      "Q776.6" { ExternalVisible := 'False'} : Bool := FALSE;   // Q776.6
      "Q776.7" { ExternalVisible := 'False'} : Bool := FALSE;   // Q776.7
      "Q777.0" { ExternalVisible := 'False'} : Bool := FALSE;   // Q777.0
      "Q777.1" { ExternalVisible := 'False'} : Bool := FALSE;   // Q777.1
      "Q777.2" { ExternalVisible := 'False'} : Bool := FALSE;   // Q777.2
      "Q777.3" { ExternalVisible := 'False'} : Bool := FALSE;   // Q777.3
      "Q777.4" { ExternalVisible := 'False'} : Bool := FALSE;   // Q777.4
      "Q777.5" { ExternalVisible := 'False'} : Bool := FALSE;   // Q777.5
      "Q777.6" { ExternalVisible := 'False'} : Bool := FALSE;   // Q777.6
      "Q777.7" { ExternalVisible := 'False'} : Bool := FALSE;   // Q777.7
      "Q778.0" { ExternalVisible := 'False'} : Bool := FALSE;   // Q778.0
      "Q778.1" { ExternalVisible := 'False'} : Bool := FALSE;   // Q778.1
      "Q778.2" { ExternalVisible := 'False'} : Bool := FALSE;   // Q778.2
      "Q778.3" { ExternalVisible := 'False'} : Bool := FALSE;   // Q778.3
      "Q778.4" { ExternalVisible := 'False'} : Bool := FALSE;   // Q778.4
      "Q778.5" { ExternalVisible := 'False'} : Bool := FALSE;   // Q778.5
      "Q778.6" { ExternalVisible := 'False'} : Bool := FALSE;   // Q778.6
      "Q778.7" { ExternalVisible := 'False'} : Bool := FALSE;   // Q778.7
      "Q779.0" { ExternalVisible := 'False'} : Bool := FALSE;   // Q779.0
      "Q779.1" { ExternalVisible := 'False'} : Bool := FALSE;   // Q779.1
      "Q779.2" { ExternalVisible := 'False'} : Bool := FALSE;   // Q779.2
      "Q779.3" { ExternalVisible := 'False'} : Bool := FALSE;   // Q779.3
      "Q779.4" { ExternalVisible := 'False'} : Bool := FALSE;   // Q779.4
      "Q779.5" { ExternalVisible := 'False'} : Bool := FALSE;   // Q779.5
      "Q779.6" { ExternalVisible := 'False'} : Bool := FALSE;   // Q779.6
      "Q779.7" { ExternalVisible := 'False'} : Bool := FALSE;   // Q779.7
      "Q780.0" { ExternalVisible := 'False'} : Bool := FALSE;   // Q780.0
      "Q780.1" { ExternalVisible := 'False'} : Bool := FALSE;   // Q780.1
      "Q780.2" { ExternalVisible := 'False'} : Bool := FALSE;   // Q780.2
      "Q780.3" { ExternalVisible := 'False'} : Bool := FALSE;   // Q780.3
      "Q780.4" { ExternalVisible := 'False'} : Bool := FALSE;   // Q780.4
      "Q780.5" { ExternalVisible := 'False'} : Bool := FALSE;   // Q780.5
      "Q780.6" { ExternalVisible := 'False'} : Bool := FALSE;   // Q780.6
      "Q780.7" { ExternalVisible := 'False'} : Bool := FALSE;   // Q780.7
      "Q781.0" { ExternalVisible := 'False'} : Bool := FALSE;   // Q781.0
      "Q781.1" { ExternalVisible := 'False'} : Bool := FALSE;   // Q781.1
      "Q781.2" { ExternalVisible := 'False'} : Bool := FALSE;   // Q781.2
      "Q781.3" { ExternalVisible := 'False'} : Bool := FALSE;   // Q781.3
      "Q781.4" { ExternalVisible := 'False'} : Bool := FALSE;   // Q781.4
      "Q781.5" { ExternalVisible := 'False'} : Bool := FALSE;   // Q781.5
      "Q781.6" { ExternalVisible := 'False'} : Bool := FALSE;   // Q781.6
      "Q781.7" { ExternalVisible := 'False'} : Bool := FALSE;   // Q781.7
      "Q782.0" { ExternalVisible := 'False'} : Bool := FALSE;   // Q782.0
      "Q782.1" { ExternalVisible := 'False'} : Bool := FALSE;   // Q782.1
      "Q782.2" { ExternalVisible := 'False'} : Bool := FALSE;   // Q782.2
      "Q782.3" { ExternalVisible := 'False'} : Bool := FALSE;   // Q782.3
      "Q782.4" { ExternalVisible := 'False'} : Bool := FALSE;   // Q782.4
      "Q782.5" { ExternalVisible := 'False'} : Bool := FALSE;   // Q782.5
      "Q782.6" { ExternalVisible := 'False'} : Bool := FALSE;   // Q782.6
      "Q782.7" { ExternalVisible := 'False'} : Bool := FALSE;   // Q782.7
      "Q783.0" { ExternalVisible := 'False'} : Bool := FALSE;   // Q783.0
      "Q783.1" { ExternalVisible := 'False'} : Bool := FALSE;   // Q783.1
      "Q783.2" { ExternalVisible := 'False'} : Bool := FALSE;   // Q783.2
      "Q783.3" { ExternalVisible := 'False'} : Bool := FALSE;   // Q783.3
      "Q783.4" { ExternalVisible := 'False'} : Bool := FALSE;   // Q783.4
      "Q783.5" { ExternalVisible := 'False'} : Bool := FALSE;   // Q783.5
      "Q783.6" { ExternalVisible := 'False'} : Bool := FALSE;   // Q783.6
      "Q783.7" { ExternalVisible := 'False'} : Bool := FALSE;   // Q783.7
      "Q784.0" { ExternalVisible := 'False'} : Bool := FALSE;   // Q784.0
      "Q784.1" { ExternalVisible := 'False'} : Bool := FALSE;   // Q784.1
      "Q784.2" { ExternalVisible := 'False'} : Bool := FALSE;   // Q784.2
      "Q784.3" { ExternalVisible := 'False'} : Bool := FALSE;   // Q784.3
      "Q784.4" { ExternalVisible := 'False'} : Bool := FALSE;   // Q784.4
      "Q784.5" { ExternalVisible := 'False'} : Bool := FALSE;   // Q784.5
      "Q784.6" { ExternalVisible := 'False'} : Bool := FALSE;   // Q784.6
      "Q784.7" { ExternalVisible := 'False'} : Bool := FALSE;   // Q784.7
      "Q785.0" { ExternalVisible := 'False'} : Bool := FALSE;   // Q785.0
      "Q785.1" { ExternalVisible := 'False'} : Bool := FALSE;   // Q785.1
      "Q785.2" { ExternalVisible := 'False'} : Bool := FALSE;   // Q785.2
      "Q785.3" { ExternalVisible := 'False'} : Bool := FALSE;   // Q785.3
      "Q785.4" { ExternalVisible := 'False'} : Bool := FALSE;   // Q785.4
      "Q785.5" { ExternalVisible := 'False'} : Bool := FALSE;   // Q785.5
      "Q785.6" { ExternalVisible := 'False'} : Bool := FALSE;   // Q785.6
      "Q785.7" { ExternalVisible := 'False'} : Bool := FALSE;   // Q785.7
      "Q786.0" { ExternalVisible := 'False'} : Bool := FALSE;   // Q786.0
      "Q786.1" { ExternalVisible := 'False'} : Bool := FALSE;   // Q786.1
      "Q786.2" { ExternalVisible := 'False'} : Bool := FALSE;   // Q786.2
      "Q786.3" { ExternalVisible := 'False'} : Bool := FALSE;   // Q786.3
      "Q786.4" { ExternalVisible := 'False'} : Bool := FALSE;   // Q786.4
      "Q786.5" { ExternalVisible := 'False'} : Bool := FALSE;   // Q786.5
      "Q786.6" { ExternalVisible := 'False'} : Bool := FALSE;   // Q786.6
      "Q786.7" { ExternalVisible := 'False'} : Bool := FALSE;   // Q786.7
      "Q787.0" { ExternalVisible := 'False'} : Bool := FALSE;   // Q787.0
      "Q787.1" { ExternalVisible := 'False'} : Bool := FALSE;   // Q787.1
      "Q787.2" { ExternalVisible := 'False'} : Bool := FALSE;   // Q787.2
      "Q787.3" { ExternalVisible := 'False'} : Bool := FALSE;   // Q787.3
      "Q787.4" { ExternalVisible := 'False'} : Bool := FALSE;   // Q787.4
      "Q787.5" { ExternalVisible := 'False'} : Bool := FALSE;   // Q787.5
      "Q787.6" { ExternalVisible := 'False'} : Bool := FALSE;   // Q787.6
      "Q787.7" { ExternalVisible := 'False'} : Bool := FALSE;   // Q787.7
      "Q788.0" { ExternalVisible := 'False'} : Bool := FALSE;   // Q788.0
      "Q788.1" { ExternalVisible := 'False'} : Bool := FALSE;   // Q788.1
      "Q788.2" { ExternalVisible := 'False'} : Bool := FALSE;   // Q788.2
      "Q788.3" { ExternalVisible := 'False'} : Bool := FALSE;   // Q788.3
      "Q788.4" { ExternalVisible := 'False'} : Bool := FALSE;   // Q788.4
      "Q788.5" { ExternalVisible := 'False'} : Bool := FALSE;   // Q788.5
      "Q788.6" { ExternalVisible := 'False'} : Bool := FALSE;   // Q788.6
      "Q788.7" { ExternalVisible := 'False'} : Bool := FALSE;   // Q788.7
      "Q789.0" { ExternalVisible := 'False'} : Bool := FALSE;   // Q789.0
      "Q789.1" { ExternalVisible := 'False'} : Bool := FALSE;   // Q789.1
      "Q789.2" { ExternalVisible := 'False'} : Bool := FALSE;   // Q789.2
      "Q789.3" { ExternalVisible := 'False'} : Bool := FALSE;   // Q789.3
      "Q789.4" { ExternalVisible := 'False'} : Bool := FALSE;   // Q789.4
      "Q789.5" { ExternalVisible := 'False'} : Bool := FALSE;   // Q789.5
      "Q789.6" { ExternalVisible := 'False'} : Bool := FALSE;   // Q789.6
      "Q789.7" { ExternalVisible := 'False'} : Bool := FALSE;   // Q789.7
      "Q790.0" { ExternalVisible := 'False'} : Bool := FALSE;   // Q790.0
      "Q790.1" { ExternalVisible := 'False'} : Bool := FALSE;   // Q790.1
      "Q790.2" { ExternalVisible := 'False'} : Bool := FALSE;   // Q790.2
      "Q790.3" { ExternalVisible := 'False'} : Bool := FALSE;   // Q790.3
      "Q790.4" { ExternalVisible := 'False'} : Bool := FALSE;   // Q790.4
      "Q790.5" { ExternalVisible := 'False'} : Bool := FALSE;   // Q790.5
      "Q790.6" { ExternalVisible := 'False'} : Bool := FALSE;   // Q790.6
      "Q790.7" { ExternalVisible := 'False'} : Bool := FALSE;   // Q790.7
      "Q791.0" { ExternalVisible := 'False'} : Bool := FALSE;   // Q791.0
      "Q791.1" { ExternalVisible := 'False'} : Bool := FALSE;   // Q791.1
      "Q791.2" { ExternalVisible := 'False'} : Bool := FALSE;   // Q791.2
      "Q791.3" { ExternalVisible := 'False'} : Bool := FALSE;   // Q791.3
      "Q791.4" { ExternalVisible := 'False'} : Bool := FALSE;   // Q791.4
      "Q791.5" { ExternalVisible := 'False'} : Bool := FALSE;   // Q791.5
      "Q791.6" { ExternalVisible := 'False'} : Bool := FALSE;   // Q791.6
      "Q791.7" { ExternalVisible := 'False'} : Bool := FALSE;   // Q791.7
      "Q792.0" { ExternalVisible := 'False'} : Bool := FALSE;   // Q792.0
      "Q792.1" { ExternalVisible := 'False'} : Bool := FALSE;   // Q792.1
      "Q792.2" { ExternalVisible := 'False'} : Bool := FALSE;   // Q792.2
      "Q792.3" { ExternalVisible := 'False'} : Bool := FALSE;   // Q792.3
      "Q792.4" { ExternalVisible := 'False'} : Bool := FALSE;   // Q792.4
      "Q792.5" { ExternalVisible := 'False'} : Bool := FALSE;   // Q792.5
      "Q792.6" { ExternalVisible := 'False'} : Bool := FALSE;   // Q792.6
      "Q792.7" { ExternalVisible := 'False'} : Bool := FALSE;   // Q792.7
      "Q793.0" { ExternalVisible := 'False'} : Bool := FALSE;   // Q793.0
      "Q793.1" { ExternalVisible := 'False'} : Bool := FALSE;   // Q793.1
      "Q793.2" { ExternalVisible := 'False'} : Bool := FALSE;   // Q793.2
      "Q793.3" { ExternalVisible := 'False'} : Bool := FALSE;   // Q793.3
      "Q793.4" { ExternalVisible := 'False'} : Bool := FALSE;   // Q793.4
      "Q793.5" { ExternalVisible := 'False'} : Bool := FALSE;   // Q793.5
      "Q793.6" { ExternalVisible := 'False'} : Bool := FALSE;   // Q793.6
      "Q793.7" { ExternalVisible := 'False'} : Bool := FALSE;   // Q793.7
      "Q794.0" { ExternalVisible := 'False'} : Bool := FALSE;   // Q794.0
      "Q794.1" { ExternalVisible := 'False'} : Bool := FALSE;   // Q794.1
      "Q794.2" { ExternalVisible := 'False'} : Bool := FALSE;   // Q794.2
      "Q794.3" { ExternalVisible := 'False'} : Bool := FALSE;   // Q794.3
      "Q794.4" { ExternalVisible := 'False'} : Bool := FALSE;   // Q794.4
      "Q794.5" { ExternalVisible := 'False'} : Bool := FALSE;   // Q794.5
      "Q794.6" { ExternalVisible := 'False'} : Bool := FALSE;   // Q794.6
      "Q794.7" { ExternalVisible := 'False'} : Bool := FALSE;   // Q794.7
      "Q795.0" { ExternalVisible := 'False'} : Bool := FALSE;   // Q795.0
      "Q795.1" { ExternalVisible := 'False'} : Bool := FALSE;   // Q795.1
      "Q795.2" { ExternalVisible := 'False'} : Bool := FALSE;   // Q795.2
      "Q795.3" { ExternalVisible := 'False'} : Bool := FALSE;   // Q795.3
      "Q795.4" { ExternalVisible := 'False'} : Bool := FALSE;   // Q795.4
      "Q795.5" { ExternalVisible := 'False'} : Bool := FALSE;   // Q795.5
      "Q795.6" { ExternalVisible := 'False'} : Bool := FALSE;   // Q795.6
      "Q795.7" { ExternalVisible := 'False'} : Bool := FALSE;   // Q795.7
      "Q796.0" { ExternalVisible := 'False'} : Bool := FALSE;   // Q796.0
      "Q796.1" { ExternalVisible := 'False'} : Bool := FALSE;   // Q796.1
      "Q796.2" { ExternalVisible := 'False'} : Bool := FALSE;   // Q796.2
      "Q796.3" { ExternalVisible := 'False'} : Bool := FALSE;   // Q796.3
      "Q796.4" { ExternalVisible := 'False'} : Bool := FALSE;   // Q796.4
      "Q796.5" { ExternalVisible := 'False'} : Bool := FALSE;   // Q796.5
      "Q796.6" { ExternalVisible := 'False'} : Bool := FALSE;   // Q796.6
      "Q796.7" { ExternalVisible := 'False'} : Bool := FALSE;   // Q796.7
      "Q797.0" { ExternalVisible := 'False'} : Bool := FALSE;   // Q797.0
      "Q797.1" { ExternalVisible := 'False'} : Bool := FALSE;   // Q797.1
      "Q797.2" { ExternalVisible := 'False'} : Bool := FALSE;   // Q797.2
      "Q797.3" { ExternalVisible := 'False'} : Bool := FALSE;   // Q797.3
      "Q797.4" { ExternalVisible := 'False'} : Bool := FALSE;   // Q797.4
      "Q797.5" { ExternalVisible := 'False'} : Bool := FALSE;   // Q797.5
      "Q797.6" { ExternalVisible := 'False'} : Bool := FALSE;   // Q797.6
      "Q797.7" { ExternalVisible := 'False'} : Bool := FALSE;   // Q797.7
      "Q798.0" { ExternalVisible := 'False'} : Bool := FALSE;   // Q798.0
      "Q798.1" { ExternalVisible := 'False'} : Bool := FALSE;   // Q798.1
      "Q798.2" { ExternalVisible := 'False'} : Bool := FALSE;   // Q798.2
      "Q798.3" { ExternalVisible := 'False'} : Bool := FALSE;   // Q798.3
      "Q798.4" { ExternalVisible := 'False'} : Bool := FALSE;   // Q798.4
      "Q798.5" { ExternalVisible := 'False'} : Bool := FALSE;   // Q798.5
      "Q798.6" { ExternalVisible := 'False'} : Bool := FALSE;   // Q798.6
      "Q798.7" { ExternalVisible := 'False'} : Bool := FALSE;   // Q798.7
      "Q799.0" { ExternalVisible := 'False'} : Bool := FALSE;   // Q799.0
      "Q799.1" { ExternalVisible := 'False'} : Bool := FALSE;   // Q799.1
      "Q799.2" { ExternalVisible := 'False'} : Bool := FALSE;   // Q799.2
      "Q799.3" { ExternalVisible := 'False'} : Bool := FALSE;   // Q799.3
      "Q799.4" { ExternalVisible := 'False'} : Bool := FALSE;   // Q799.4
      "Q799.5" { ExternalVisible := 'False'} : Bool := FALSE;   // Q799.5
      "Q799.6" { ExternalVisible := 'False'} : Bool := FALSE;   // Q799.6
      "Q799.7" { ExternalVisible := 'False'} : Bool := FALSE;   // Q799.7
      "Q800.0" { ExternalVisible := 'False'} : Bool := FALSE;   // Q800.0
      "Q800.1" { ExternalVisible := 'False'} : Bool := FALSE;   // Q800.1
      "Q800.2" { ExternalVisible := 'False'} : Bool := FALSE;   // Q800.2
      "Q800.3" { ExternalVisible := 'False'} : Bool := FALSE;   // Q800.3
      "Q800.4" { ExternalVisible := 'False'} : Bool := FALSE;   // Q800.4
      "Q800.5" { ExternalVisible := 'False'} : Bool := FALSE;   // Q800.5
      "Q800.6" { ExternalVisible := 'False'} : Bool := FALSE;   // Q800.6
      "Q800.7" { ExternalVisible := 'False'} : Bool := FALSE;   // Q800.7
      "Q801.0" { ExternalVisible := 'False'} : Bool := FALSE;   // Q801.0
      "Q801.1" { ExternalVisible := 'False'} : Bool := FALSE;   // Q801.1
      "Q801.2" { ExternalVisible := 'False'} : Bool := FALSE;   // Q801.2
      "Q801.3" { ExternalVisible := 'False'} : Bool := FALSE;   // Q801.3
      "Q801.4" { ExternalVisible := 'False'} : Bool := FALSE;   // Q801.4
      "Q801.5" { ExternalVisible := 'False'} : Bool := FALSE;   // Q801.5
      "Q801.6" { ExternalVisible := 'False'} : Bool := FALSE;   // Q801.6
      "Q801.7" { ExternalVisible := 'False'} : Bool := FALSE;   // Q801.7
      "Q802.0" { ExternalVisible := 'False'} : Bool := FALSE;   // Q802.0
      "Q802.1" { ExternalVisible := 'False'} : Bool := FALSE;   // Q802.1
      "Q802.2" { ExternalVisible := 'False'} : Bool := FALSE;   // Q802.2
      "Q802.3" { ExternalVisible := 'False'} : Bool := FALSE;   // Q802.3
      "Q802.4" { ExternalVisible := 'False'} : Bool := FALSE;   // Q802.4
      "Q802.5" { ExternalVisible := 'False'} : Bool := FALSE;   // Q802.5
      "Q802.6" { ExternalVisible := 'False'} : Bool := FALSE;   // Q802.6
      "Q802.7" { ExternalVisible := 'False'} : Bool := FALSE;   // Q802.7
      "Q803.0" { ExternalVisible := 'False'} : Bool := FALSE;   // Q803.0
      "Q803.1" { ExternalVisible := 'False'} : Bool := FALSE;   // Q803.1
      "Q803.2" { ExternalVisible := 'False'} : Bool := FALSE;   // Q803.2
      "Q803.3" { ExternalVisible := 'False'} : Bool := FALSE;   // Q803.3
      "Q803.4" { ExternalVisible := 'False'} : Bool := FALSE;   // Q803.4
      "Q803.5" { ExternalVisible := 'False'} : Bool := FALSE;   // Q803.5
      "Q803.6" { ExternalVisible := 'False'} : Bool := FALSE;   // Q803.6
      "Q803.7" { ExternalVisible := 'False'} : Bool := FALSE;   // Q803.7
      "Q804.0" { ExternalVisible := 'False'} : Bool := FALSE;   // Q804.0
      "Q804.1" { ExternalVisible := 'False'} : Bool := FALSE;   // Q804.1
      "Q804.2" { ExternalVisible := 'False'} : Bool := FALSE;   // Q804.2
      "Q804.3" { ExternalVisible := 'False'} : Bool := FALSE;   // Q804.3
      "Q804.4" { ExternalVisible := 'False'} : Bool := FALSE;   // Q804.4
      "Q804.5" { ExternalVisible := 'False'} : Bool := FALSE;   // Q804.5
      "Q804.6" { ExternalVisible := 'False'} : Bool := FALSE;   // Q804.6
      "Q804.7" { ExternalVisible := 'False'} : Bool := FALSE;   // Q804.7
      "Q805.0" { ExternalVisible := 'False'} : Bool := FALSE;   // Q805.0
      "Q805.1" { ExternalVisible := 'False'} : Bool := FALSE;   // Q805.1
      "Q805.2" { ExternalVisible := 'False'} : Bool := FALSE;   // Q805.2
      "Q805.3" { ExternalVisible := 'False'} : Bool := FALSE;   // Q805.3
      "Q805.4" { ExternalVisible := 'False'} : Bool := FALSE;   // Q805.4
      "Q805.5" { ExternalVisible := 'False'} : Bool := FALSE;   // Q805.5
      "Q805.6" { ExternalVisible := 'False'} : Bool := FALSE;   // Q805.6
      "Q805.7" { ExternalVisible := 'False'} : Bool := FALSE;   // Q805.7
      "Q806.0" { ExternalVisible := 'False'} : Bool := FALSE;   // Q806.0
      "Q806.1" { ExternalVisible := 'False'} : Bool := FALSE;   // Q806.1
      "Q806.2" { ExternalVisible := 'False'} : Bool := FALSE;   // Q806.2
      "Q806.3" { ExternalVisible := 'False'} : Bool := FALSE;   // Q806.3
      "Q806.4" { ExternalVisible := 'False'} : Bool := FALSE;   // Q806.4
      "Q806.5" { ExternalVisible := 'False'} : Bool := FALSE;   // Q806.5
      "Q806.6" { ExternalVisible := 'False'} : Bool := FALSE;   // Q806.6
      "Q806.7" { ExternalVisible := 'False'} : Bool := FALSE;   // Q806.7
      "Q807.0" { ExternalVisible := 'False'} : Bool := FALSE;   // Q807.0
      "Q807.1" { ExternalVisible := 'False'} : Bool := FALSE;   // Q807.1
      "Q807.2" { ExternalVisible := 'False'} : Bool := FALSE;   // Q807.2
      "Q807.3" { ExternalVisible := 'False'} : Bool := FALSE;   // Q807.3
      "Q807.4" { ExternalVisible := 'False'} : Bool := FALSE;   // Q807.4
      "Q807.5" { ExternalVisible := 'False'} : Bool := FALSE;   // Q807.5
      "Q807.6" { ExternalVisible := 'False'} : Bool := FALSE;   // Q807.6
      "Q807.7" { ExternalVisible := 'False'} : Bool := FALSE;   // Q807.7
      "Q808.0" { ExternalVisible := 'False'} : Bool := FALSE;   // Q808.0
      "Q808.1" { ExternalVisible := 'False'} : Bool := FALSE;   // Q808.1
      "Q808.2" { ExternalVisible := 'False'} : Bool := FALSE;   // Q808.2
      "Q808.3" { ExternalVisible := 'False'} : Bool := FALSE;   // Q808.3
      "Q808.4" { ExternalVisible := 'False'} : Bool := FALSE;   // Q808.4
      "Q808.5" { ExternalVisible := 'False'} : Bool := FALSE;   // Q808.5
      "Q808.6" { ExternalVisible := 'False'} : Bool := FALSE;   // Q808.6
      "Q808.7" { ExternalVisible := 'False'} : Bool := FALSE;   // Q808.7
      "Q809.0" { ExternalVisible := 'False'} : Bool := FALSE;   // Q809.0
      "Q809.1" { ExternalVisible := 'False'} : Bool := FALSE;   // Q809.1
      "Q809.2" { ExternalVisible := 'False'} : Bool := FALSE;   // Q809.2
      "Q809.3" { ExternalVisible := 'False'} : Bool := FALSE;   // Q809.3
      "Q809.4" { ExternalVisible := 'False'} : Bool := FALSE;   // Q809.4
      "Q809.5" { ExternalVisible := 'False'} : Bool := FALSE;   // Q809.5
      "Q809.6" { ExternalVisible := 'False'} : Bool := FALSE;   // Q809.6
      "Q809.7" { ExternalVisible := 'False'} : Bool := FALSE;   // Q809.7
      "Q810.0" { ExternalVisible := 'False'} : Bool := FALSE;   // Q810.0
      "Q810.1" { ExternalVisible := 'False'} : Bool := FALSE;   // Q810.1
      "Q810.2" { ExternalVisible := 'False'} : Bool := FALSE;   // Q810.2
      "Q810.3" { ExternalVisible := 'False'} : Bool := FALSE;   // Q810.3
      "Q810.4" { ExternalVisible := 'False'} : Bool := FALSE;   // Q810.4
      "Q810.5" { ExternalVisible := 'False'} : Bool := FALSE;   // Q810.5
      "Q810.6" { ExternalVisible := 'False'} : Bool := FALSE;   // Q810.6
      "Q810.7" { ExternalVisible := 'False'} : Bool := FALSE;   // Q810.7
      "Q811.0" { ExternalVisible := 'False'} : Bool := FALSE;   // Q811.0
      "Q811.1" { ExternalVisible := 'False'} : Bool := FALSE;   // Q811.1
      "Q811.2" { ExternalVisible := 'False'} : Bool := FALSE;   // Q811.2
      "Q811.3" { ExternalVisible := 'False'} : Bool := FALSE;   // Q811.3
      "Q811.4" { ExternalVisible := 'False'} : Bool := FALSE;   // Q811.4
      "Q811.5" { ExternalVisible := 'False'} : Bool := FALSE;   // Q811.5
      "Q811.6" { ExternalVisible := 'False'} : Bool := FALSE;   // Q811.6
      "Q811.7" { ExternalVisible := 'False'} : Bool := FALSE;   // Q811.7
      "Q812.0" { ExternalVisible := 'False'} : Bool := FALSE;   // Q812.0
      "Q812.1" { ExternalVisible := 'False'} : Bool := FALSE;   // Q812.1
      "Q812.2" { ExternalVisible := 'False'} : Bool := FALSE;   // Q812.2
      "Q812.3" { ExternalVisible := 'False'} : Bool := FALSE;   // Q812.3
      "Q812.4" { ExternalVisible := 'False'} : Bool := FALSE;   // Q812.4
      "Q812.5" { ExternalVisible := 'False'} : Bool := FALSE;   // Q812.5
      "Q812.6" { ExternalVisible := 'False'} : Bool := FALSE;   // Q812.6
      "Q812.7" { ExternalVisible := 'False'} : Bool := FALSE;   // Q812.7
      "Q813.0" { ExternalVisible := 'False'} : Bool := FALSE;   // Q813.0
      "Q813.1" { ExternalVisible := 'False'} : Bool := FALSE;   // Q813.1
      "Q813.2" { ExternalVisible := 'False'} : Bool := FALSE;   // Q813.2
      "Q813.3" { ExternalVisible := 'False'} : Bool := FALSE;   // Q813.3
      "Q813.4" { ExternalVisible := 'False'} : Bool := FALSE;   // Q813.4
      "Q813.5" { ExternalVisible := 'False'} : Bool := FALSE;   // Q813.5
      "Q813.6" { ExternalVisible := 'False'} : Bool := FALSE;   // Q813.6
      "Q813.7" { ExternalVisible := 'False'} : Bool := FALSE;   // Q813.7
      "Q814.0" { ExternalVisible := 'False'} : Bool := FALSE;   // Q814.0
      "Q814.1" { ExternalVisible := 'False'} : Bool := FALSE;   // Q814.1
      "Q814.2" { ExternalVisible := 'False'} : Bool := FALSE;   // Q814.2
      "Q814.3" { ExternalVisible := 'False'} : Bool := FALSE;   // Q814.3
      "Q814.4" { ExternalVisible := 'False'} : Bool := FALSE;   // Q814.4
      "Q814.5" { ExternalVisible := 'False'} : Bool := FALSE;   // Q814.5
      "Q814.6" { ExternalVisible := 'False'} : Bool := FALSE;   // Q814.6
      "Q814.7" { ExternalVisible := 'False'} : Bool := FALSE;   // Q814.7
      "Q815.0" { ExternalVisible := 'False'} : Bool := FALSE;   // Q815.0
      "Q815.1" { ExternalVisible := 'False'} : Bool := FALSE;   // Q815.1
      "Q815.2" { ExternalVisible := 'False'} : Bool := FALSE;   // Q815.2
      "Q815.3" { ExternalVisible := 'False'} : Bool := FALSE;   // Q815.3
      "Q815.4" { ExternalVisible := 'False'} : Bool := FALSE;   // Q815.4
      "Q815.5" { ExternalVisible := 'False'} : Bool := FALSE;   // Q815.5
      "Q815.6" { ExternalVisible := 'False'} : Bool := FALSE;   // Q815.6
      "Q815.7" { ExternalVisible := 'False'} : Bool := FALSE;   // Q815.7
      "Q816.0" { ExternalVisible := 'False'} : Bool := FALSE;   // Q816.0
      "Q816.1" { ExternalVisible := 'False'} : Bool := FALSE;   // Q816.1
      "Q816.2" { ExternalVisible := 'False'} : Bool := FALSE;   // Q816.2
      "Q816.3" { ExternalVisible := 'False'} : Bool := FALSE;   // Q816.3
      "Q816.4" { ExternalVisible := 'False'} : Bool := FALSE;   // Q816.4
      "Q816.5" { ExternalVisible := 'False'} : Bool := FALSE;   // Q816.5
      "Q816.6" { ExternalVisible := 'False'} : Bool := FALSE;   // Q816.6
      "Q816.7" { ExternalVisible := 'False'} : Bool := FALSE;   // Q816.7
      "Q817.0" { ExternalVisible := 'False'} : Bool := FALSE;   // Q817.0
      "Q817.1" { ExternalVisible := 'False'} : Bool := FALSE;   // Q817.1
      "Q817.2" { ExternalVisible := 'False'} : Bool := FALSE;   // Q817.2
      "Q817.3" { ExternalVisible := 'False'} : Bool := FALSE;   // Q817.3
      "Q817.4" { ExternalVisible := 'False'} : Bool := FALSE;   // Q817.4
      "Q817.5" { ExternalVisible := 'False'} : Bool := FALSE;   // Q817.5
      "Q817.6" { ExternalVisible := 'False'} : Bool := FALSE;   // Q817.6
      "Q817.7" { ExternalVisible := 'False'} : Bool := FALSE;   // Q817.7
      "Q818.0" { ExternalVisible := 'False'} : Bool := FALSE;   // Q818.0
      "Q818.1" { ExternalVisible := 'False'} : Bool := FALSE;   // Q818.1
      "Q818.2" { ExternalVisible := 'False'} : Bool := FALSE;   // Q818.2
      "Q818.3" { ExternalVisible := 'False'} : Bool := FALSE;   // Q818.3
      "Q818.4" { ExternalVisible := 'False'} : Bool := FALSE;   // Q818.4
      "Q818.5" { ExternalVisible := 'False'} : Bool := FALSE;   // Q818.5
      "Q818.6" { ExternalVisible := 'False'} : Bool := FALSE;   // Q818.6
      "Q818.7" { ExternalVisible := 'False'} : Bool := FALSE;   // Q818.7
      "Q819.0" { ExternalVisible := 'False'} : Bool := FALSE;   // Q819.0
      "Q819.1" { ExternalVisible := 'False'} : Bool := FALSE;   // Q819.1
      "Q819.2" { ExternalVisible := 'False'} : Bool := FALSE;   // Q819.2
      "Q819.3" { ExternalVisible := 'False'} : Bool := FALSE;   // Q819.3
      "Q819.4" { ExternalVisible := 'False'} : Bool := FALSE;   // Q819.4
      "Q819.5" { ExternalVisible := 'False'} : Bool := FALSE;   // Q819.5
      "Q819.6" { ExternalVisible := 'False'} : Bool := FALSE;   // Q819.6
      "Q819.7" { ExternalVisible := 'False'} : Bool := FALSE;   // Q819.7
      "Q820.0" { ExternalVisible := 'False'} : Bool := FALSE;   // Q820.0
      "Q820.1" { ExternalVisible := 'False'} : Bool := FALSE;   // Q820.1
      "Q820.2" { ExternalVisible := 'False'} : Bool := FALSE;   // Q820.2
      "Q820.3" { ExternalVisible := 'False'} : Bool := FALSE;   // Q820.3
      "Q820.4" { ExternalVisible := 'False'} : Bool := FALSE;   // Q820.4
      "Q820.5" { ExternalVisible := 'False'} : Bool := FALSE;   // Q820.5
      "Q820.6" { ExternalVisible := 'False'} : Bool := FALSE;   // Q820.6
      "Q820.7" { ExternalVisible := 'False'} : Bool := FALSE;   // Q820.7
      "Q821.0" { ExternalVisible := 'False'} : Bool := FALSE;   // Q821.0
      "Q821.1" { ExternalVisible := 'False'} : Bool := FALSE;   // Q821.1
      "Q821.2" { ExternalVisible := 'False'} : Bool := FALSE;   // Q821.2
      "Q821.3" { ExternalVisible := 'False'} : Bool := FALSE;   // Q821.3
      "Q821.4" { ExternalVisible := 'False'} : Bool := FALSE;   // Q821.4
      "Q821.5" { ExternalVisible := 'False'} : Bool := FALSE;   // Q821.5
      "Q821.6" { ExternalVisible := 'False'} : Bool := FALSE;   // Q821.6
      "Q821.7" { ExternalVisible := 'False'} : Bool := FALSE;   // Q821.7
      "Q822.0" { ExternalVisible := 'False'} : Bool := FALSE;   // Q822.0
      "Q822.1" { ExternalVisible := 'False'} : Bool := FALSE;   // Q822.1
      "Q822.2" { ExternalVisible := 'False'} : Bool := FALSE;   // Q822.2
      "Q822.3" { ExternalVisible := 'False'} : Bool := FALSE;   // Q822.3
      "Q822.4" { ExternalVisible := 'False'} : Bool := FALSE;   // Q822.4
      "Q822.5" { ExternalVisible := 'False'} : Bool := FALSE;   // Q822.5
      "Q822.6" { ExternalVisible := 'False'} : Bool := FALSE;   // Q822.6
      "Q822.7" { ExternalVisible := 'False'} : Bool := FALSE;   // Q822.7
      "Q823.0" { ExternalVisible := 'False'} : Bool := FALSE;   // Q823.0
      "Q823.1" { ExternalVisible := 'False'} : Bool := FALSE;   // Q823.1
      "Q823.2" { ExternalVisible := 'False'} : Bool := FALSE;   // Q823.2
      "Q823.3" { ExternalVisible := 'False'} : Bool := FALSE;   // Q823.3
      "Q823.4" { ExternalVisible := 'False'} : Bool := FALSE;   // Q823.4
      "Q823.5" { ExternalVisible := 'False'} : Bool := FALSE;   // Q823.5
      "Q823.6" { ExternalVisible := 'False'} : Bool := FALSE;   // Q823.6
      "Q823.7" { ExternalVisible := 'False'} : Bool := FALSE;   // Q823.7
      "Q824.0" { ExternalVisible := 'False'} : Bool := FALSE;   // Q824.0
      "Q824.1" { ExternalVisible := 'False'} : Bool := FALSE;   // Q824.1
      "Q824.2" { ExternalVisible := 'False'} : Bool := FALSE;   // Q824.2
      "Q824.3" { ExternalVisible := 'False'} : Bool := FALSE;   // Q824.3
      "Q824.4" { ExternalVisible := 'False'} : Bool := FALSE;   // Q824.4
      "Q824.5" { ExternalVisible := 'False'} : Bool := FALSE;   // Q824.5
      "Q824.6" { ExternalVisible := 'False'} : Bool := FALSE;   // Q824.6
      "Q824.7" { ExternalVisible := 'False'} : Bool := FALSE;   // Q824.7
      "Q825.0" { ExternalVisible := 'False'} : Bool := FALSE;   // Q825.0
      "Q825.1" { ExternalVisible := 'False'} : Bool := FALSE;   // Q825.1
      "Q825.2" { ExternalVisible := 'False'} : Bool := FALSE;   // Q825.2
      "Q825.3" { ExternalVisible := 'False'} : Bool := FALSE;   // Q825.3
      "Q825.4" { ExternalVisible := 'False'} : Bool := FALSE;   // Q825.4
      "Q825.5" { ExternalVisible := 'False'} : Bool := FALSE;   // Q825.5
      "Q825.6" { ExternalVisible := 'False'} : Bool := FALSE;   // Q825.6
      "Q825.7" { ExternalVisible := 'False'} : Bool := FALSE;   // Q825.7
      "Q826.0" { ExternalVisible := 'False'} : Bool := FALSE;   // Q826.0
      "Q826.1" { ExternalVisible := 'False'} : Bool := FALSE;   // Q826.1
      "Q826.2" { ExternalVisible := 'False'} : Bool := FALSE;   // Q826.2
      "Q826.3" { ExternalVisible := 'False'} : Bool := FALSE;   // Q826.3
      "Q826.4" { ExternalVisible := 'False'} : Bool := FALSE;   // Q826.4
      "Q826.5" { ExternalVisible := 'False'} : Bool := FALSE;   // Q826.5
      "Q826.6" { ExternalVisible := 'False'} : Bool := FALSE;   // Q826.6
      "Q826.7" { ExternalVisible := 'False'} : Bool := FALSE;   // Q826.7
      "Q827.0" { ExternalVisible := 'False'} : Bool := FALSE;   // Q827.0
      "Q827.1" { ExternalVisible := 'False'} : Bool := FALSE;   // Q827.1
      "Q827.2" { ExternalVisible := 'False'} : Bool := FALSE;   // Q827.2
      "Q827.3" { ExternalVisible := 'False'} : Bool := FALSE;   // Q827.3
      "Q827.4" { ExternalVisible := 'False'} : Bool := FALSE;   // Q827.4
      "Q827.5" { ExternalVisible := 'False'} : Bool := FALSE;   // Q827.5
      "Q827.6" { ExternalVisible := 'False'} : Bool := FALSE;   // Q827.6
      "Q827.7" { ExternalVisible := 'False'} : Bool := FALSE;   // Q827.7
      "Q828.0" { ExternalVisible := 'False'} : Bool := FALSE;   // Q828.0
      "Q828.1" { ExternalVisible := 'False'} : Bool := FALSE;   // Q828.1
      "Q828.2" { ExternalVisible := 'False'} : Bool := FALSE;   // Q828.2
      "Q828.3" { ExternalVisible := 'False'} : Bool := FALSE;   // Q828.3
      "Q828.4" { ExternalVisible := 'False'} : Bool := FALSE;   // Q828.4
      "Q828.5" { ExternalVisible := 'False'} : Bool := FALSE;   // Q828.5
      "Q828.6" { ExternalVisible := 'False'} : Bool := FALSE;   // Q828.6
      "Q828.7" { ExternalVisible := 'False'} : Bool := FALSE;   // Q828.7
      "Q829.0" { ExternalVisible := 'False'} : Bool := FALSE;   // Q829.0
      "Q829.1" { ExternalVisible := 'False'} : Bool := FALSE;   // Q829.1
      "Q829.2" { ExternalVisible := 'False'} : Bool := FALSE;   // Q829.2
      "Q829.3" { ExternalVisible := 'False'} : Bool := FALSE;   // Q829.3
      "Q829.4" { ExternalVisible := 'False'} : Bool := FALSE;   // Q829.4
      "Q829.5" { ExternalVisible := 'False'} : Bool := FALSE;   // Q829.5
      "Q829.6" { ExternalVisible := 'False'} : Bool := FALSE;   // Q829.6
      "Q829.7" { ExternalVisible := 'False'} : Bool := FALSE;   // Q829.7
      "Q830.0" { ExternalVisible := 'False'} : Bool := FALSE;   // Q830.0
      "Q830.1" { ExternalVisible := 'False'} : Bool := FALSE;   // Q830.1
      "Q830.2" { ExternalVisible := 'False'} : Bool := FALSE;   // Q830.2
      "Q830.3" { ExternalVisible := 'False'} : Bool := FALSE;   // Q830.3
      "Q830.4" { ExternalVisible := 'False'} : Bool := FALSE;   // Q830.4
      "Q830.5" { ExternalVisible := 'False'} : Bool := FALSE;   // Q830.5
      "Q830.6" { ExternalVisible := 'False'} : Bool := FALSE;   // Q830.6
      "Q830.7" { ExternalVisible := 'False'} : Bool := FALSE;   // Q830.7
      "Q831.0" { ExternalVisible := 'False'} : Bool := FALSE;   // Q831.0
      "Q831.1" { ExternalVisible := 'False'} : Bool := FALSE;   // Q831.1
      "Q831.2" { ExternalVisible := 'False'} : Bool := FALSE;   // Q831.2
      "Q831.3" { ExternalVisible := 'False'} : Bool := FALSE;   // Q831.3
      "Q831.4" { ExternalVisible := 'False'} : Bool := FALSE;   // Q831.4
      "Q831.5" { ExternalVisible := 'False'} : Bool := FALSE;   // Q831.5
      "Q831.6" { ExternalVisible := 'False'} : Bool := FALSE;   // Q831.6
      "Q831.7" { ExternalVisible := 'False'} : Bool := FALSE;   // Q831.7
      "Q832.0" { ExternalVisible := 'False'} : Bool := FALSE;   // Q832.0
      "Q832.1" { ExternalVisible := 'False'} : Bool := FALSE;   // Q832.1
      "Q832.2" { ExternalVisible := 'False'} : Bool := FALSE;   // Q832.2
      "Q832.3" { ExternalVisible := 'False'} : Bool := FALSE;   // Q832.3
      "Q832.4" { ExternalVisible := 'False'} : Bool := FALSE;   // Q832.4
      "Q832.5" { ExternalVisible := 'False'} : Bool := FALSE;   // Q832.5
      "Q832.6" { ExternalVisible := 'False'} : Bool := FALSE;   // Q832.6
      "Q832.7" { ExternalVisible := 'False'} : Bool := FALSE;   // Q832.7
      "Q833.0" { ExternalVisible := 'False'} : Bool := FALSE;   // Q833.0
      "Q833.1" { ExternalVisible := 'False'} : Bool := FALSE;   // Q833.1
      "Q833.2" { ExternalVisible := 'False'} : Bool := FALSE;   // Q833.2
      "Q833.3" { ExternalVisible := 'False'} : Bool := FALSE;   // Q833.3
      "Q833.4" { ExternalVisible := 'False'} : Bool := FALSE;   // Q833.4
      "Q833.5" { ExternalVisible := 'False'} : Bool := FALSE;   // Q833.5
      "Q833.6" { ExternalVisible := 'False'} : Bool := FALSE;   // Q833.6
      "Q833.7" { ExternalVisible := 'False'} : Bool := FALSE;   // Q833.7
      "Q834.0" { ExternalVisible := 'False'} : Bool := FALSE;   // Q834.0
      "Q834.1" { ExternalVisible := 'False'} : Bool := FALSE;   // Q834.1
      "Q834.2" { ExternalVisible := 'False'} : Bool := FALSE;   // Q834.2
      "Q834.3" { ExternalVisible := 'False'} : Bool := FALSE;   // Q834.3
      "Q834.4" { ExternalVisible := 'False'} : Bool := FALSE;   // Q834.4
      "Q834.5" { ExternalVisible := 'False'} : Bool := FALSE;   // Q834.5
      "Q834.6" { ExternalVisible := 'False'} : Bool := FALSE;   // Q834.6
      "Q834.7" { ExternalVisible := 'False'} : Bool := FALSE;   // Q834.7
      "Q835.0" { ExternalVisible := 'False'} : Bool := FALSE;   // Q835.0
      "Q835.1" { ExternalVisible := 'False'} : Bool := FALSE;   // Q835.1
      "Q835.2" { ExternalVisible := 'False'} : Bool := FALSE;   // Q835.2
      "Q835.3" { ExternalVisible := 'False'} : Bool := FALSE;   // Q835.3
      "Q835.4" { ExternalVisible := 'False'} : Bool := FALSE;   // Q835.4
      "Q835.5" { ExternalVisible := 'False'} : Bool := FALSE;   // Q835.5
      "Q835.6" { ExternalVisible := 'False'} : Bool := FALSE;   // Q835.6
      "Q835.7" { ExternalVisible := 'False'} : Bool := FALSE;   // Q835.7
      "Q836.0" { ExternalVisible := 'False'} : Bool := FALSE;   // Q836.0
      "Q836.1" { ExternalVisible := 'False'} : Bool := FALSE;   // Q836.1
      "Q836.2" { ExternalVisible := 'False'} : Bool := FALSE;   // Q836.2
      "Q836.3" { ExternalVisible := 'False'} : Bool := FALSE;   // Q836.3
      "Q836.4" { ExternalVisible := 'False'} : Bool := FALSE;   // Q836.4
      "Q836.5" { ExternalVisible := 'False'} : Bool := FALSE;   // Q836.5
      "Q836.6" { ExternalVisible := 'False'} : Bool := FALSE;   // Q836.6
      "Q836.7" { ExternalVisible := 'False'} : Bool := FALSE;   // Q836.7
      "Q837.0" { ExternalVisible := 'False'} : Bool := FALSE;   // Q837.0
      "Q837.1" { ExternalVisible := 'False'} : Bool := FALSE;   // Q837.1
      "Q837.2" { ExternalVisible := 'False'} : Bool := FALSE;   // Q837.2
      "Q837.3" { ExternalVisible := 'False'} : Bool := FALSE;   // Q837.3
      "Q837.4" { ExternalVisible := 'False'} : Bool := FALSE;   // Q837.4
      "Q837.5" { ExternalVisible := 'False'} : Bool := FALSE;   // Q837.5
      "Q837.6" { ExternalVisible := 'False'} : Bool := FALSE;   // Q837.6
      "Q837.7" { ExternalVisible := 'False'} : Bool := FALSE;   // Q837.7
      "Q838.0" { ExternalVisible := 'False'} : Bool := FALSE;   // Q838.0
      "Q838.1" { ExternalVisible := 'False'} : Bool := FALSE;   // Q838.1
      "Q838.2" { ExternalVisible := 'False'} : Bool := FALSE;   // Q838.2
      "Q838.3" { ExternalVisible := 'False'} : Bool := FALSE;   // Q838.3
      "Q838.4" { ExternalVisible := 'False'} : Bool := FALSE;   // Q838.4
      "Q838.5" { ExternalVisible := 'False'} : Bool := FALSE;   // Q838.5
      "Q838.6" { ExternalVisible := 'False'} : Bool := FALSE;   // Q838.6
      "Q838.7" { ExternalVisible := 'False'} : Bool := FALSE;   // Q838.7
      "Q839.0" { ExternalVisible := 'False'} : Bool := FALSE;   // Q839.0
      "Q839.1" { ExternalVisible := 'False'} : Bool := FALSE;   // Q839.1
      "Q839.2" { ExternalVisible := 'False'} : Bool := FALSE;   // Q839.2
      "Q839.3" { ExternalVisible := 'False'} : Bool := FALSE;   // Q839.3
      "Q839.4" { ExternalVisible := 'False'} : Bool := FALSE;   // Q839.4
      "Q839.5" { ExternalVisible := 'False'} : Bool := FALSE;   // Q839.5
      "Q839.6" { ExternalVisible := 'False'} : Bool := FALSE;   // Q839.6
      "Q839.7" { ExternalVisible := 'False'} : Bool := FALSE;   // Q839.7
      "Q840.0" { ExternalVisible := 'False'} : Bool := FALSE;   // Q840.0
      "Q840.1" { ExternalVisible := 'False'} : Bool := FALSE;   // Q840.1
      "Q840.2" { ExternalVisible := 'False'} : Bool := FALSE;   // Q840.2
      "Q840.3" { ExternalVisible := 'False'} : Bool := FALSE;   // Q840.3
      "Q840.4" { ExternalVisible := 'False'} : Bool := FALSE;   // Q840.4
      "Q840.5" { ExternalVisible := 'False'} : Bool := FALSE;   // Q840.5
      "Q840.6" { ExternalVisible := 'False'} : Bool := FALSE;   // Q840.6
      "Q840.7" { ExternalVisible := 'False'} : Bool := FALSE;   // Q840.7
      "Q841.0" { ExternalVisible := 'False'} : Bool := FALSE;   // Q841.0
      "Q841.1" { ExternalVisible := 'False'} : Bool := FALSE;   // Q841.1
      "Q841.2" { ExternalVisible := 'False'} : Bool := FALSE;   // Q841.2
      "Q841.3" { ExternalVisible := 'False'} : Bool := FALSE;   // Q841.3
      "Q841.4" { ExternalVisible := 'False'} : Bool := FALSE;   // Q841.4
      "Q841.5" { ExternalVisible := 'False'} : Bool := FALSE;   // Q841.5
      "Q841.6" { ExternalVisible := 'False'} : Bool := FALSE;   // Q841.6
      "Q841.7" { ExternalVisible := 'False'} : Bool := FALSE;   // Q841.7
      "Q842.0" { ExternalVisible := 'False'} : Bool := FALSE;   // Q842.0
      "Q842.1" { ExternalVisible := 'False'} : Bool := FALSE;   // Q842.1
      "Q842.2" { ExternalVisible := 'False'} : Bool := FALSE;   // Q842.2
      "Q842.3" { ExternalVisible := 'False'} : Bool := FALSE;   // Q842.3
      "Q842.4" { ExternalVisible := 'False'} : Bool := FALSE;   // Q842.4
      "Q842.5" { ExternalVisible := 'False'} : Bool := FALSE;   // Q842.5
      "Q842.6" { ExternalVisible := 'False'} : Bool := FALSE;   // Q842.6
      "Q842.7" { ExternalVisible := 'False'} : Bool := FALSE;   // Q842.7
      "Q843.0" { ExternalVisible := 'False'} : Bool := FALSE;   // Q843.0
      "Q843.1" { ExternalVisible := 'False'} : Bool := FALSE;   // Q843.1
      "Q843.2" { ExternalVisible := 'False'} : Bool := FALSE;   // Q843.2
      "Q843.3" { ExternalVisible := 'False'} : Bool := FALSE;   // Q843.3
      "Q843.4" { ExternalVisible := 'False'} : Bool := FALSE;   // Q843.4
      "Q843.5" { ExternalVisible := 'False'} : Bool := FALSE;   // Q843.5
      "Q843.6" { ExternalVisible := 'False'} : Bool := FALSE;   // Q843.6
      "Q843.7" { ExternalVisible := 'False'} : Bool := FALSE;   // Q843.7
      "Q844.0" { ExternalVisible := 'False'} : Bool := FALSE;   // Q844.0
      "Q844.1" { ExternalVisible := 'False'} : Bool := FALSE;   // Q844.1
      "Q844.2" { ExternalVisible := 'False'} : Bool := FALSE;   // Q844.2
      "Q844.3" { ExternalVisible := 'False'} : Bool := FALSE;   // Q844.3
      "Q844.4" { ExternalVisible := 'False'} : Bool := FALSE;   // Q844.4
      "Q844.5" { ExternalVisible := 'False'} : Bool := FALSE;   // Q844.5
      "Q844.6" { ExternalVisible := 'False'} : Bool := FALSE;   // Q844.6
      "Q844.7" { ExternalVisible := 'False'} : Bool := FALSE;   // Q844.7
      "Q845.0" { ExternalVisible := 'False'} : Bool := FALSE;   // Q845.0
      "Q845.1" { ExternalVisible := 'False'} : Bool := FALSE;   // Q845.1
      "Q845.2" { ExternalVisible := 'False'} : Bool := FALSE;   // Q845.2
      "Q845.3" { ExternalVisible := 'False'} : Bool := FALSE;   // Q845.3
      "Q845.4" { ExternalVisible := 'False'} : Bool := FALSE;   // Q845.4
      "Q845.5" { ExternalVisible := 'False'} : Bool := FALSE;   // Q845.5
      "Q845.6" { ExternalVisible := 'False'} : Bool := FALSE;   // Q845.6
      "Q845.7" { ExternalVisible := 'False'} : Bool := FALSE;   // Q845.7
      "Q846.0" { ExternalVisible := 'False'} : Bool := FALSE;   // Q846.0
      "Q846.1" { ExternalVisible := 'False'} : Bool := FALSE;   // Q846.1
      "Q846.2" { ExternalVisible := 'False'} : Bool := FALSE;   // Q846.2
      "Q846.3" { ExternalVisible := 'False'} : Bool := FALSE;   // Q846.3
      "Q846.4" { ExternalVisible := 'False'} : Bool := FALSE;   // Q846.4
      "Q846.5" { ExternalVisible := 'False'} : Bool := FALSE;   // Q846.5
      "Q846.6" { ExternalVisible := 'False'} : Bool := FALSE;   // Q846.6
      "Q846.7" { ExternalVisible := 'False'} : Bool := FALSE;   // Q846.7
      "Q847.0" { ExternalVisible := 'False'} : Bool := FALSE;   // Q847.0
      "Q847.1" { ExternalVisible := 'False'} : Bool := FALSE;   // Q847.1
      "Q847.2" { ExternalVisible := 'False'} : Bool := FALSE;   // Q847.2
      "Q847.3" { ExternalVisible := 'False'} : Bool := FALSE;   // Q847.3
      "Q847.4" { ExternalVisible := 'False'} : Bool := FALSE;   // Q847.4
      "Q847.5" { ExternalVisible := 'False'} : Bool := FALSE;   // Q847.5
      "Q847.6" { ExternalVisible := 'False'} : Bool := FALSE;   // Q847.6
      "Q847.7" { ExternalVisible := 'False'} : Bool := FALSE;   // Q847.7
      "Q848.0" { ExternalVisible := 'False'} : Bool := FALSE;   // Q848.0
      "Q848.1" { ExternalVisible := 'False'} : Bool := FALSE;   // Q848.1
      "Q848.2" { ExternalVisible := 'False'} : Bool := FALSE;   // Q848.2
      "Q848.3" { ExternalVisible := 'False'} : Bool := FALSE;   // Q848.3
      "Q848.4" { ExternalVisible := 'False'} : Bool := FALSE;   // Q848.4
      "Q848.5" { ExternalVisible := 'False'} : Bool := FALSE;   // Q848.5
      "Q848.6" { ExternalVisible := 'False'} : Bool := FALSE;   // Q848.6
      "Q848.7" { ExternalVisible := 'False'} : Bool := FALSE;   // Q848.7
      "Q849.0" { ExternalVisible := 'False'} : Bool := FALSE;   // Q849.0
      "Q849.1" { ExternalVisible := 'False'} : Bool := FALSE;   // Q849.1
      "Q849.2" { ExternalVisible := 'False'} : Bool := FALSE;   // Q849.2
      "Q849.3" { ExternalVisible := 'False'} : Bool := FALSE;   // Q849.3
      "Q849.4" { ExternalVisible := 'False'} : Bool := FALSE;   // Q849.4
      "Q849.5" { ExternalVisible := 'False'} : Bool := FALSE;   // Q849.5
      "Q849.6" { ExternalVisible := 'False'} : Bool := FALSE;   // Q849.6
      "Q849.7" { ExternalVisible := 'False'} : Bool := FALSE;   // Q849.7
      "Q850.0" { ExternalVisible := 'False'} : Bool := FALSE;   // Q850.0
      "Q850.1" { ExternalVisible := 'False'} : Bool := FALSE;   // Q850.1
      "Q850.2" { ExternalVisible := 'False'} : Bool := FALSE;   // Q850.2
      "Q850.3" { ExternalVisible := 'False'} : Bool := FALSE;   // Q850.3
      "Q850.4" { ExternalVisible := 'False'} : Bool := FALSE;   // Q850.4
      "Q850.5" { ExternalVisible := 'False'} : Bool := FALSE;   // Q850.5
      "Q850.6" { ExternalVisible := 'False'} : Bool := FALSE;   // Q850.6
      "Q850.7" { ExternalVisible := 'False'} : Bool := FALSE;   // Q850.7
      "Q851.0" { ExternalVisible := 'False'} : Bool := FALSE;   // Q851.0
      "Q851.1" { ExternalVisible := 'False'} : Bool := FALSE;   // Q851.1
      "Q851.2" { ExternalVisible := 'False'} : Bool := FALSE;   // Q851.2
      "Q851.3" { ExternalVisible := 'False'} : Bool := FALSE;   // Q851.3
      "Q851.4" { ExternalVisible := 'False'} : Bool := FALSE;   // Q851.4
      "Q851.5" { ExternalVisible := 'False'} : Bool := FALSE;   // Q851.5
      "Q851.6" { ExternalVisible := 'False'} : Bool := FALSE;   // Q851.6
      "Q851.7" { ExternalVisible := 'False'} : Bool := FALSE;   // Q851.7
      "Q852.0" { ExternalVisible := 'False'} : Bool := FALSE;   // Q852.0
      "Q852.1" { ExternalVisible := 'False'} : Bool := FALSE;   // Q852.1
      "Q852.2" { ExternalVisible := 'False'} : Bool := FALSE;   // Q852.2
      "Q852.3" { ExternalVisible := 'False'} : Bool := FALSE;   // Q852.3
      "Q852.4" { ExternalVisible := 'False'} : Bool := FALSE;   // Q852.4
      "Q852.5" { ExternalVisible := 'False'} : Bool := FALSE;   // Q852.5
      "Q852.6" { ExternalVisible := 'False'} : Bool := FALSE;   // Q852.6
      "Q852.7" { ExternalVisible := 'False'} : Bool := FALSE;   // Q852.7
      "Q853.0" { ExternalVisible := 'False'} : Bool := FALSE;   // Q853.0
      "Q853.1" { ExternalVisible := 'False'} : Bool := FALSE;   // Q853.1
      "Q853.2" { ExternalVisible := 'False'} : Bool := FALSE;   // Q853.2
      "Q853.3" { ExternalVisible := 'False'} : Bool := FALSE;   // Q853.3
      "Q853.4" { ExternalVisible := 'False'} : Bool := FALSE;   // Q853.4
      "Q853.5" { ExternalVisible := 'False'} : Bool := FALSE;   // Q853.5
      "Q853.6" { ExternalVisible := 'False'} : Bool := FALSE;   // Q853.6
      "Q853.7" { ExternalVisible := 'False'} : Bool := FALSE;   // Q853.7
      "Q854.0" { ExternalVisible := 'False'} : Bool := FALSE;   // Q854.0
      "Q854.1" { ExternalVisible := 'False'} : Bool := FALSE;   // Q854.1
      "Q854.2" { ExternalVisible := 'False'} : Bool := FALSE;   // Q854.2
      "Q854.3" { ExternalVisible := 'False'} : Bool := FALSE;   // Q854.3
      "Q854.4" { ExternalVisible := 'False'} : Bool := FALSE;   // Q854.4
      "Q854.5" { ExternalVisible := 'False'} : Bool := FALSE;   // Q854.5
      "Q854.6" { ExternalVisible := 'False'} : Bool := FALSE;   // Q854.6
      "Q854.7" { ExternalVisible := 'False'} : Bool := FALSE;   // Q854.7
      "Q855.0" { ExternalVisible := 'False'} : Bool := FALSE;   // Q855.0
      "Q855.1" { ExternalVisible := 'False'} : Bool := FALSE;   // Q855.1
      "Q855.2" { ExternalVisible := 'False'} : Bool := FALSE;   // Q855.2
      "Q855.3" { ExternalVisible := 'False'} : Bool := FALSE;   // Q855.3
      "Q855.4" { ExternalVisible := 'False'} : Bool := FALSE;   // Q855.4
      "Q855.5" { ExternalVisible := 'False'} : Bool := FALSE;   // Q855.5
      "Q855.6" { ExternalVisible := 'False'} : Bool := FALSE;   // Q855.6
      "Q855.7" { ExternalVisible := 'False'} : Bool := FALSE;   // Q855.7
      "Q856.0" { ExternalVisible := 'False'} : Bool := FALSE;   // Q856.0
      "Q856.1" { ExternalVisible := 'False'} : Bool := FALSE;   // Q856.1
      "Q856.2" { ExternalVisible := 'False'} : Bool := FALSE;   // Q856.2
      "Q856.3" { ExternalVisible := 'False'} : Bool := FALSE;   // Q856.3
      "Q856.4" { ExternalVisible := 'False'} : Bool := FALSE;   // Q856.4
      "Q856.5" { ExternalVisible := 'False'} : Bool := FALSE;   // Q856.5
      "Q856.6" { ExternalVisible := 'False'} : Bool := FALSE;   // Q856.6
      "Q856.7" { ExternalVisible := 'False'} : Bool := FALSE;   // Q856.7
      "Q857.0" { ExternalVisible := 'False'} : Bool := FALSE;   // Q857.0
      "Q857.1" { ExternalVisible := 'False'} : Bool := FALSE;   // Q857.1
      "Q857.2" { ExternalVisible := 'False'} : Bool := FALSE;   // Q857.2
      "Q857.3" { ExternalVisible := 'False'} : Bool := FALSE;   // Q857.3
      "Q857.4" { ExternalVisible := 'False'} : Bool := FALSE;   // Q857.4
      "Q857.5" { ExternalVisible := 'False'} : Bool := FALSE;   // Q857.5
      "Q857.6" { ExternalVisible := 'False'} : Bool := FALSE;   // Q857.6
      "Q857.7" { ExternalVisible := 'False'} : Bool := FALSE;   // Q857.7
      "Q858.0" { ExternalVisible := 'False'} : Bool := FALSE;   // Q858.0
      "Q858.1" { ExternalVisible := 'False'} : Bool := FALSE;   // Q858.1
      "Q858.2" { ExternalVisible := 'False'} : Bool := FALSE;   // Q858.2
      "Q858.3" { ExternalVisible := 'False'} : Bool := FALSE;   // Q858.3
      "Q858.4" { ExternalVisible := 'False'} : Bool := FALSE;   // Q858.4
      "Q858.5" { ExternalVisible := 'False'} : Bool := FALSE;   // Q858.5
      "Q858.6" { ExternalVisible := 'False'} : Bool := FALSE;   // Q858.6
      "Q858.7" { ExternalVisible := 'False'} : Bool := FALSE;   // Q858.7
      "Q859.0" { ExternalVisible := 'False'} : Bool := FALSE;   // Q859.0
      "Q859.1" { ExternalVisible := 'False'} : Bool := FALSE;   // Q859.1
      "Q859.2" { ExternalVisible := 'False'} : Bool := FALSE;   // Q859.2
      "Q859.3" { ExternalVisible := 'False'} : Bool := FALSE;   // Q859.3
      "Q859.4" { ExternalVisible := 'False'} : Bool := FALSE;   // Q859.4
      "Q859.5" { ExternalVisible := 'False'} : Bool := FALSE;   // Q859.5
      "Q859.6" { ExternalVisible := 'False'} : Bool := FALSE;   // Q859.6
      "Q859.7" { ExternalVisible := 'False'} : Bool := FALSE;   // Q859.7
      "Q860.0" { ExternalVisible := 'False'} : Bool := FALSE;   // Q860.0
      "Q860.1" { ExternalVisible := 'False'} : Bool := FALSE;   // Q860.1
      "Q860.2" { ExternalVisible := 'False'} : Bool := FALSE;   // Q860.2
      "Q860.3" { ExternalVisible := 'False'} : Bool := FALSE;   // Q860.3
      "Q860.4" { ExternalVisible := 'False'} : Bool := FALSE;   // Q860.4
      "Q860.5" { ExternalVisible := 'False'} : Bool := FALSE;   // Q860.5
      "Q860.6" { ExternalVisible := 'False'} : Bool := FALSE;   // Q860.6
      "Q860.7" { ExternalVisible := 'False'} : Bool := FALSE;   // Q860.7
      "Q861.0" { ExternalVisible := 'False'} : Bool := FALSE;   // Q861.0
      "Q861.1" { ExternalVisible := 'False'} : Bool := FALSE;   // Q861.1
      "Q861.2" { ExternalVisible := 'False'} : Bool := FALSE;   // Q861.2
      "Q861.3" { ExternalVisible := 'False'} : Bool := FALSE;   // Q861.3
      "Q861.4" { ExternalVisible := 'False'} : Bool := FALSE;   // Q861.4
      "Q861.5" { ExternalVisible := 'False'} : Bool := FALSE;   // Q861.5
      "Q861.6" { ExternalVisible := 'False'} : Bool := FALSE;   // Q861.6
      "Q861.7" { ExternalVisible := 'False'} : Bool := FALSE;   // Q861.7
      "Q862.0" { ExternalVisible := 'False'} : Bool := FALSE;   // Q862.0
      "Q862.1" { ExternalVisible := 'False'} : Bool := FALSE;   // Q862.1
      "Q862.2" { ExternalVisible := 'False'} : Bool := FALSE;   // Q862.2
      "Q862.3" { ExternalVisible := 'False'} : Bool := FALSE;   // Q862.3
      "Q862.4" { ExternalVisible := 'False'} : Bool := FALSE;   // Q862.4
      "Q862.5" { ExternalVisible := 'False'} : Bool := FALSE;   // Q862.5
      "Q862.6" { ExternalVisible := 'False'} : Bool := FALSE;   // Q862.6
      "Q862.7" { ExternalVisible := 'False'} : Bool := FALSE;   // Q862.7
      "Q863.0" { ExternalVisible := 'False'} : Bool := FALSE;   // Q863.0
      "Q863.1" { ExternalVisible := 'False'} : Bool := FALSE;   // Q863.1
      "Q863.2" { ExternalVisible := 'False'} : Bool := FALSE;   // Q863.2
      "Q863.3" { ExternalVisible := 'False'} : Bool := FALSE;   // Q863.3
      "Q863.4" { ExternalVisible := 'False'} : Bool := FALSE;   // Q863.4
      "Q863.5" { ExternalVisible := 'False'} : Bool := FALSE;   // Q863.5
      "Q863.6" { ExternalVisible := 'False'} : Bool := FALSE;   // Q863.6
      "Q863.7" { ExternalVisible := 'False'} : Bool := FALSE;   // Q863.7
      "Q864.0" { ExternalVisible := 'False'} : Bool := FALSE;   // Q864.0
      "Q864.1" { ExternalVisible := 'False'} : Bool := FALSE;   // Q864.1
      "Q864.2" { ExternalVisible := 'False'} : Bool := FALSE;   // Q864.2
      "Q864.3" { ExternalVisible := 'False'} : Bool := FALSE;   // Q864.3
      "Q864.4" { ExternalVisible := 'False'} : Bool := FALSE;   // Q864.4
      "Q864.5" { ExternalVisible := 'False'} : Bool := FALSE;   // Q864.5
      "Q864.6" { ExternalVisible := 'False'} : Bool := FALSE;   // Q864.6
      "Q864.7" { ExternalVisible := 'False'} : Bool := FALSE;   // Q864.7
      "Q865.0" { ExternalVisible := 'False'} : Bool := FALSE;   // Q865.0
      "Q865.1" { ExternalVisible := 'False'} : Bool := FALSE;   // Q865.1
      "Q865.2" { ExternalVisible := 'False'} : Bool := FALSE;   // Q865.2
      "Q865.3" { ExternalVisible := 'False'} : Bool := FALSE;   // Q865.3
      "Q865.4" { ExternalVisible := 'False'} : Bool := FALSE;   // Q865.4
      "Q865.5" { ExternalVisible := 'False'} : Bool := FALSE;   // Q865.5
      "Q865.6" { ExternalVisible := 'False'} : Bool := FALSE;   // Q865.6
      "Q865.7" { ExternalVisible := 'False'} : Bool := FALSE;   // Q865.7
      "Q866.0" { ExternalVisible := 'False'} : Bool := FALSE;   // Q866.0
      "Q866.1" { ExternalVisible := 'False'} : Bool := FALSE;   // Q866.1
      "Q866.2" { ExternalVisible := 'False'} : Bool := FALSE;   // Q866.2
      "Q866.3" { ExternalVisible := 'False'} : Bool := FALSE;   // Q866.3
      "Q866.4" { ExternalVisible := 'False'} : Bool := FALSE;   // Q866.4
      "Q866.5" { ExternalVisible := 'False'} : Bool := FALSE;   // Q866.5
      "Q866.6" { ExternalVisible := 'False'} : Bool := FALSE;   // Q866.6
      "Q866.7" { ExternalVisible := 'False'} : Bool := FALSE;   // Q866.7
      "Q867.0" { ExternalVisible := 'False'} : Bool := FALSE;   // Q867.0
      "Q867.1" { ExternalVisible := 'False'} : Bool := FALSE;   // Q867.1
      "Q867.2" { ExternalVisible := 'False'} : Bool := FALSE;   // Q867.2
      "Q867.3" { ExternalVisible := 'False'} : Bool := FALSE;   // Q867.3
      "Q867.4" { ExternalVisible := 'False'} : Bool := FALSE;   // Q867.4
      "Q867.5" { ExternalVisible := 'False'} : Bool := FALSE;   // Q867.5
      "Q867.6" { ExternalVisible := 'False'} : Bool := FALSE;   // Q867.6
      "Q867.7" { ExternalVisible := 'False'} : Bool := FALSE;   // Q867.7
      "Q868.0" { ExternalVisible := 'False'} : Bool := FALSE;   // Q868.0
      "Q868.1" { ExternalVisible := 'False'} : Bool := FALSE;   // Q868.1
      "Q868.2" { ExternalVisible := 'False'} : Bool := FALSE;   // Q868.2
      "Q868.3" { ExternalVisible := 'False'} : Bool := FALSE;   // Q868.3
      "Q868.4" { ExternalVisible := 'False'} : Bool := FALSE;   // Q868.4
      "Q868.5" { ExternalVisible := 'False'} : Bool := FALSE;   // Q868.5
      "Q868.6" { ExternalVisible := 'False'} : Bool := FALSE;   // Q868.6
      "Q868.7" { ExternalVisible := 'False'} : Bool := FALSE;   // Q868.7
      "Q869.0" { ExternalVisible := 'False'} : Bool := FALSE;   // Q869.0
      "Q869.1" { ExternalVisible := 'False'} : Bool := FALSE;   // Q869.1
      "Q869.2" { ExternalVisible := 'False'} : Bool := FALSE;   // Q869.2
      "Q869.3" { ExternalVisible := 'False'} : Bool := FALSE;   // Q869.3
      "Q869.4" { ExternalVisible := 'False'} : Bool := FALSE;   // Q869.4
      "Q869.5" { ExternalVisible := 'False'} : Bool := FALSE;   // Q869.5
      "Q869.6" { ExternalVisible := 'False'} : Bool := FALSE;   // Q869.6
      "Q869.7" { ExternalVisible := 'False'} : Bool := FALSE;   // Q869.7
      "Q870.0" { ExternalVisible := 'False'} : Bool := FALSE;   // Q870.0
      "Q870.1" { ExternalVisible := 'False'} : Bool := FALSE;   // Q870.1
      "Q870.2" { ExternalVisible := 'False'} : Bool := FALSE;   // Q870.2
      "Q870.3" { ExternalVisible := 'False'} : Bool := FALSE;   // Q870.3
      "Q870.4" { ExternalVisible := 'False'} : Bool := FALSE;   // Q870.4
      "Q870.5" { ExternalVisible := 'False'} : Bool := FALSE;   // Q870.5
      "Q870.6" { ExternalVisible := 'False'} : Bool := FALSE;   // Q870.6
      "Q870.7" { ExternalVisible := 'False'} : Bool := FALSE;   // Q870.7
      "Q871.0" { ExternalVisible := 'False'} : Bool := FALSE;   // Q871.0
      "Q871.1" { ExternalVisible := 'False'} : Bool := FALSE;   // Q871.1
      "Q871.2" { ExternalVisible := 'False'} : Bool := FALSE;   // Q871.2
      "Q871.3" { ExternalVisible := 'False'} : Bool := FALSE;   // Q871.3
      "Q871.4" { ExternalVisible := 'False'} : Bool := FALSE;   // Q871.4
      "Q871.5" { ExternalVisible := 'False'} : Bool := FALSE;   // Q871.5
      "Q871.6" { ExternalVisible := 'False'} : Bool := FALSE;   // Q871.6
      "Q871.7" { ExternalVisible := 'False'} : Bool := FALSE;   // Q871.7
      "Q872.0" { ExternalVisible := 'False'} : Bool := FALSE;   // Q872.0
      "Q872.1" { ExternalVisible := 'False'} : Bool := FALSE;   // Q872.1
      "Q872.2" { ExternalVisible := 'False'} : Bool := FALSE;   // Q872.2
      "Q872.3" { ExternalVisible := 'False'} : Bool := FALSE;   // Q872.3
      "Q872.4" { ExternalVisible := 'False'} : Bool := FALSE;   // Q872.4
      "Q872.5" { ExternalVisible := 'False'} : Bool := FALSE;   // Q872.5
      "Q872.6" { ExternalVisible := 'False'} : Bool := FALSE;   // Q872.6
      "Q872.7" { ExternalVisible := 'False'} : Bool := FALSE;   // Q872.7
      "Q873.0" { ExternalVisible := 'False'} : Bool := FALSE;   // Q873.0
      "Q873.1" { ExternalVisible := 'False'} : Bool := FALSE;   // Q873.1
      "Q873.2" { ExternalVisible := 'False'} : Bool := FALSE;   // Q873.2
      "Q873.3" { ExternalVisible := 'False'} : Bool := FALSE;   // Q873.3
      "Q873.4" { ExternalVisible := 'False'} : Bool := FALSE;   // Q873.4
      "Q873.5" { ExternalVisible := 'False'} : Bool := FALSE;   // Q873.5
      "Q873.6" { ExternalVisible := 'False'} : Bool := FALSE;   // Q873.6
      "Q873.7" { ExternalVisible := 'False'} : Bool := FALSE;   // Q873.7
      "Q874.0" { ExternalVisible := 'False'} : Bool := FALSE;   // Q874.0
      "Q874.1" { ExternalVisible := 'False'} : Bool := FALSE;   // Q874.1
      "Q874.2" { ExternalVisible := 'False'} : Bool := FALSE;   // Q874.2
      "Q874.3" { ExternalVisible := 'False'} : Bool := FALSE;   // Q874.3
      "Q874.4" { ExternalVisible := 'False'} : Bool := FALSE;   // Q874.4
      "Q874.5" { ExternalVisible := 'False'} : Bool := FALSE;   // Q874.5
      "Q874.6" { ExternalVisible := 'False'} : Bool := FALSE;   // Q874.6
      "Q874.7" { ExternalVisible := 'False'} : Bool := FALSE;   // Q874.7
      "Q875.0" { ExternalVisible := 'False'} : Bool := FALSE;   // Q875.0
      "Q875.1" { ExternalVisible := 'False'} : Bool := FALSE;   // Q875.1
      "Q875.2" { ExternalVisible := 'False'} : Bool := FALSE;   // Q875.2
      "Q875.3" { ExternalVisible := 'False'} : Bool := FALSE;   // Q875.3
      "Q875.4" { ExternalVisible := 'False'} : Bool := FALSE;   // Q875.4
      "Q875.5" { ExternalVisible := 'False'} : Bool := FALSE;   // Q875.5
      "Q875.6" { ExternalVisible := 'False'} : Bool := FALSE;   // Q875.6
      "Q875.7" { ExternalVisible := 'False'} : Bool := FALSE;   // Q875.7
      "Q876.0" { ExternalVisible := 'False'} : Bool := FALSE;   // Q876.0
      "Q876.1" { ExternalVisible := 'False'} : Bool := FALSE;   // Q876.1
      "Q876.2" { ExternalVisible := 'False'} : Bool := FALSE;   // Q876.2
      "Q876.3" { ExternalVisible := 'False'} : Bool := FALSE;   // Q876.3
      "Q876.4" { ExternalVisible := 'False'} : Bool := FALSE;   // Q876.4
      "Q876.5" { ExternalVisible := 'False'} : Bool := FALSE;   // Q876.5
      "Q876.6" { ExternalVisible := 'False'} : Bool := FALSE;   // Q876.6
      "Q876.7" { ExternalVisible := 'False'} : Bool := FALSE;   // Q876.7
      "Q877.0" { ExternalVisible := 'False'} : Bool := FALSE;   // Q877.0
      "Q877.1" { ExternalVisible := 'False'} : Bool := FALSE;   // Q877.1
      "Q877.2" { ExternalVisible := 'False'} : Bool := FALSE;   // Q877.2
      "Q877.3" { ExternalVisible := 'False'} : Bool := FALSE;   // Q877.3
      "Q877.4" { ExternalVisible := 'False'} : Bool := FALSE;   // Q877.4
      "Q877.5" { ExternalVisible := 'False'} : Bool := FALSE;   // Q877.5
      "Q877.6" { ExternalVisible := 'False'} : Bool := FALSE;   // Q877.6
      "Q877.7" { ExternalVisible := 'False'} : Bool := FALSE;   // Q877.7
      "Q878.0" { ExternalVisible := 'False'} : Bool := FALSE;   // Q878.0
      "Q878.1" { ExternalVisible := 'False'} : Bool := FALSE;   // Q878.1
      "Q878.2" { ExternalVisible := 'False'} : Bool := FALSE;   // Q878.2
      "Q878.3" { ExternalVisible := 'False'} : Bool := FALSE;   // Q878.3
      "Q878.4" { ExternalVisible := 'False'} : Bool := FALSE;   // Q878.4
      "Q878.5" { ExternalVisible := 'False'} : Bool := FALSE;   // Q878.5
      "Q878.6" { ExternalVisible := 'False'} : Bool := FALSE;   // Q878.6
      "Q878.7" { ExternalVisible := 'False'} : Bool := FALSE;   // Q878.7
      "Q879.0" { ExternalVisible := 'False'} : Bool := FALSE;   // Q879.0
      "Q879.1" { ExternalVisible := 'False'} : Bool := FALSE;   // Q879.1
      "Q879.2" { ExternalVisible := 'False'} : Bool := FALSE;   // Q879.2
      "Q879.3" { ExternalVisible := 'False'} : Bool := FALSE;   // Q879.3
      "Q879.4" { ExternalVisible := 'False'} : Bool := FALSE;   // Q879.4
      "Q879.5" { ExternalVisible := 'False'} : Bool := FALSE;   // Q879.5
      "Q879.6" { ExternalVisible := 'False'} : Bool := FALSE;   // Q879.6
      "Q879.7" { ExternalVisible := 'False'} : Bool := FALSE;   // Q879.7
      "Q880.0" { ExternalVisible := 'False'} : Bool := FALSE;   // Q880.0
      "Q880.1" { ExternalVisible := 'False'} : Bool := FALSE;   // Q880.1
      "Q880.2" { ExternalVisible := 'False'} : Bool := FALSE;   // Q880.2
      "Q880.3" { ExternalVisible := 'False'} : Bool := FALSE;   // Q880.3
      "Q880.4" { ExternalVisible := 'False'} : Bool := FALSE;   // Q880.4
      "Q880.5" { ExternalVisible := 'False'} : Bool := FALSE;   // Q880.5
      "Q880.6" { ExternalVisible := 'False'} : Bool := FALSE;   // Q880.6
      "Q880.7" { ExternalVisible := 'False'} : Bool := FALSE;   // Q880.7
      "Q881.0" { ExternalVisible := 'False'} : Bool := FALSE;   // Q881.0
      "Q881.1" { ExternalVisible := 'False'} : Bool := FALSE;   // Q881.1
      "Q881.2" { ExternalVisible := 'False'} : Bool := FALSE;   // Q881.2
      "Q881.3" { ExternalVisible := 'False'} : Bool := FALSE;   // Q881.3
      "Q881.4" { ExternalVisible := 'False'} : Bool := FALSE;   // Q881.4
      "Q881.5" { ExternalVisible := 'False'} : Bool := FALSE;   // Q881.5
      "Q881.6" { ExternalVisible := 'False'} : Bool := FALSE;   // Q881.6
      "Q881.7" { ExternalVisible := 'False'} : Bool := FALSE;   // Q881.7
      "Q882.0" { ExternalVisible := 'False'} : Bool := FALSE;   // Q882.0
      "Q882.1" { ExternalVisible := 'False'} : Bool := FALSE;   // Q882.1
      "Q882.2" { ExternalVisible := 'False'} : Bool := FALSE;   // Q882.2
      "Q882.3" { ExternalVisible := 'False'} : Bool := FALSE;   // Q882.3
      "Q882.4" { ExternalVisible := 'False'} : Bool := FALSE;   // Q882.4
      "Q882.5" { ExternalVisible := 'False'} : Bool := FALSE;   // Q882.5
      "Q882.6" { ExternalVisible := 'False'} : Bool := FALSE;   // Q882.6
      "Q882.7" { ExternalVisible := 'False'} : Bool := FALSE;   // Q882.7
      "Q883.0" { ExternalVisible := 'False'} : Bool := FALSE;   // Q883.0
      "Q883.1" { ExternalVisible := 'False'} : Bool := FALSE;   // Q883.1
      "Q883.2" { ExternalVisible := 'False'} : Bool := FALSE;   // Q883.2
      "Q883.3" { ExternalVisible := 'False'} : Bool := FALSE;   // Q883.3
      "Q883.4" { ExternalVisible := 'False'} : Bool := FALSE;   // Q883.4
      "Q883.5" { ExternalVisible := 'False'} : Bool := FALSE;   // Q883.5
      "Q883.6" { ExternalVisible := 'False'} : Bool := FALSE;   // Q883.6
      "Q883.7" { ExternalVisible := 'False'} : Bool := FALSE;   // Q883.7
      "Q884.0" { ExternalVisible := 'False'} : Bool := FALSE;   // Q884.0
      "Q884.1" { ExternalVisible := 'False'} : Bool := FALSE;   // Q884.1
      "Q884.2" { ExternalVisible := 'False'} : Bool := FALSE;   // Q884.2
      "Q884.3" { ExternalVisible := 'False'} : Bool := FALSE;   // Q884.3
      "Q884.4" { ExternalVisible := 'False'} : Bool := FALSE;   // Q884.4
      "Q884.5" { ExternalVisible := 'False'} : Bool := FALSE;   // Q884.5
      "Q884.6" { ExternalVisible := 'False'} : Bool := FALSE;   // Q884.6
      "Q884.7" { ExternalVisible := 'False'} : Bool := FALSE;   // Q884.7
      "Q885.0" { ExternalVisible := 'False'} : Bool := FALSE;   // Q885.0
      "Q885.1" { ExternalVisible := 'False'} : Bool := FALSE;   // Q885.1
      "Q885.2" { ExternalVisible := 'False'} : Bool := FALSE;   // Q885.2
      "Q885.3" { ExternalVisible := 'False'} : Bool := FALSE;   // Q885.3
      "Q885.4" { ExternalVisible := 'False'} : Bool := FALSE;   // Q885.4
      "Q885.5" { ExternalVisible := 'False'} : Bool := FALSE;   // Q885.5
      "Q885.6" { ExternalVisible := 'False'} : Bool := FALSE;   // Q885.6
      "Q885.7" { ExternalVisible := 'False'} : Bool := FALSE;   // Q885.7
      "Q886.0" { ExternalVisible := 'False'} : Bool := FALSE;   // Q886.0
      "Q886.1" { ExternalVisible := 'False'} : Bool := FALSE;   // Q886.1
      "Q886.2" { ExternalVisible := 'False'} : Bool := FALSE;   // Q886.2
      "Q886.3" { ExternalVisible := 'False'} : Bool := FALSE;   // Q886.3
      "Q886.4" { ExternalVisible := 'False'} : Bool := FALSE;   // Q886.4
      "Q886.5" { ExternalVisible := 'False'} : Bool := FALSE;   // Q886.5
      "Q886.6" { ExternalVisible := 'False'} : Bool := FALSE;   // Q886.6
      "Q886.7" { ExternalVisible := 'False'} : Bool := FALSE;   // Q886.7
      "Q887.0" { ExternalVisible := 'False'} : Bool := FALSE;   // Q887.0
      "Q887.1" { ExternalVisible := 'False'} : Bool := FALSE;   // Q887.1
      "Q887.2" { ExternalVisible := 'False'} : Bool := FALSE;   // Q887.2
      "Q887.3" { ExternalVisible := 'False'} : Bool := FALSE;   // Q887.3
      "Q887.4" { ExternalVisible := 'False'} : Bool := FALSE;   // Q887.4
      "Q887.5" { ExternalVisible := 'False'} : Bool := FALSE;   // Q887.5
      "Q887.6" { ExternalVisible := 'False'} : Bool := FALSE;   // Q887.6
      "Q887.7" { ExternalVisible := 'False'} : Bool := FALSE;   // Q887.7
      "Q888.0" { ExternalVisible := 'False'} : Bool := FALSE;   // Q888.0
      "Q888.1" { ExternalVisible := 'False'} : Bool := FALSE;   // Q888.1
      "Q888.2" { ExternalVisible := 'False'} : Bool := FALSE;   // Q888.2
      "Q888.3" { ExternalVisible := 'False'} : Bool := FALSE;   // Q888.3
      "Q888.4" { ExternalVisible := 'False'} : Bool := FALSE;   // Q888.4
      "Q888.5" { ExternalVisible := 'False'} : Bool := FALSE;   // Q888.5
      "Q888.6" { ExternalVisible := 'False'} : Bool := FALSE;   // Q888.6
      "Q888.7" { ExternalVisible := 'False'} : Bool := FALSE;   // Q888.7
      "Q889.0" { ExternalVisible := 'False'} : Bool := FALSE;   // Q889.0
      "Q889.1" { ExternalVisible := 'False'} : Bool := FALSE;   // Q889.1
      "Q889.2" { ExternalVisible := 'False'} : Bool := FALSE;   // Q889.2
      "Q889.3" { ExternalVisible := 'False'} : Bool := FALSE;   // Q889.3
      "Q889.4" { ExternalVisible := 'False'} : Bool := FALSE;   // Q889.4
      "Q889.5" { ExternalVisible := 'False'} : Bool := FALSE;   // Q889.5
      "Q889.6" { ExternalVisible := 'False'} : Bool := FALSE;   // Q889.6
      "Q889.7" { ExternalVisible := 'False'} : Bool := FALSE;   // Q889.7
      "Q890.0" { ExternalVisible := 'False'} : Bool := FALSE;   // Q890.0
      "Q890.1" { ExternalVisible := 'False'} : Bool := FALSE;   // Q890.1
      "Q890.2" { ExternalVisible := 'False'} : Bool := FALSE;   // Q890.2
      "Q890.3" { ExternalVisible := 'False'} : Bool := FALSE;   // Q890.3
      "Q890.4" { ExternalVisible := 'False'} : Bool := FALSE;   // Q890.4
      "Q890.5" { ExternalVisible := 'False'} : Bool := FALSE;   // Q890.5
      "Q890.6" { ExternalVisible := 'False'} : Bool := FALSE;   // Q890.6
      "Q890.7" { ExternalVisible := 'False'} : Bool := FALSE;   // Q890.7
      "Q891.0" { ExternalVisible := 'False'} : Bool := FALSE;   // Q891.0
      "Q891.1" { ExternalVisible := 'False'} : Bool := FALSE;   // Q891.1
      "Q891.2" { ExternalVisible := 'False'} : Bool := FALSE;   // Q891.2
      "Q891.3" { ExternalVisible := 'False'} : Bool := FALSE;   // Q891.3
      "Q891.4" { ExternalVisible := 'False'} : Bool := FALSE;   // Q891.4
      "Q891.5" { ExternalVisible := 'False'} : Bool := FALSE;   // Q891.5
      "Q891.6" { ExternalVisible := 'False'} : Bool := FALSE;   // Q891.6
      "Q891.7" { ExternalVisible := 'False'} : Bool := FALSE;   // Q891.7
      "Q892.0" { ExternalVisible := 'False'} : Bool := FALSE;   // Q892.0
      "Q892.1" { ExternalVisible := 'False'} : Bool := FALSE;   // Q892.1
      "Q892.2" { ExternalVisible := 'False'} : Bool := FALSE;   // Q892.2
      "Q892.3" { ExternalVisible := 'False'} : Bool := FALSE;   // Q892.3
      "Q892.4" { ExternalVisible := 'False'} : Bool := FALSE;   // Q892.4
      "Q892.5" { ExternalVisible := 'False'} : Bool := FALSE;   // Q892.5
      "Q892.6" { ExternalVisible := 'False'} : Bool := FALSE;   // Q892.6
      "Q892.7" { ExternalVisible := 'False'} : Bool := FALSE;   // Q892.7
      "Q893.0" { ExternalVisible := 'False'} : Bool := FALSE;   // Q893.0
      "Q893.1" { ExternalVisible := 'False'} : Bool := FALSE;   // Q893.1
      "Q893.2" { ExternalVisible := 'False'} : Bool := FALSE;   // Q893.2
      "Q893.3" { ExternalVisible := 'False'} : Bool := FALSE;   // Q893.3
      "Q893.4" { ExternalVisible := 'False'} : Bool := FALSE;   // Q893.4
      "Q893.5" { ExternalVisible := 'False'} : Bool := FALSE;   // Q893.5
      "Q893.6" { ExternalVisible := 'False'} : Bool := FALSE;   // Q893.6
      "Q893.7" { ExternalVisible := 'False'} : Bool := FALSE;   // Q893.7
      "Q894.0" { ExternalVisible := 'False'} : Bool := FALSE;   // Q894.0
      "Q894.1" { ExternalVisible := 'False'} : Bool := FALSE;   // Q894.1
      "Q894.2" { ExternalVisible := 'False'} : Bool := FALSE;   // Q894.2
      "Q894.3" { ExternalVisible := 'False'} : Bool := FALSE;   // Q894.3
      "Q894.4" { ExternalVisible := 'False'} : Bool := FALSE;   // Q894.4
      "Q894.5" { ExternalVisible := 'False'} : Bool := FALSE;   // Q894.5
      "Q894.6" { ExternalVisible := 'False'} : Bool := FALSE;   // Q894.6
      "Q894.7" { ExternalVisible := 'False'} : Bool := FALSE;   // Q894.7
      "Q895.0" { ExternalVisible := 'False'} : Bool := FALSE;   // Q895.0
      "Q895.1" { ExternalVisible := 'False'} : Bool := FALSE;   // Q895.1
      "Q895.2" { ExternalVisible := 'False'} : Bool := FALSE;   // Q895.2
      "Q895.3" { ExternalVisible := 'False'} : Bool := FALSE;   // Q895.3
      "Q895.4" { ExternalVisible := 'False'} : Bool := FALSE;   // Q895.4
      "Q895.5" { ExternalVisible := 'False'} : Bool := FALSE;   // Q895.5
      "Q895.6" { ExternalVisible := 'False'} : Bool := FALSE;   // Q895.6
      "Q895.7" { ExternalVisible := 'False'} : Bool := FALSE;   // Q895.7
      "Q896.0" { ExternalVisible := 'False'} : Bool := FALSE;   // Q896.0
      "Q896.1" { ExternalVisible := 'False'} : Bool := FALSE;   // Q896.1
      "Q896.2" { ExternalVisible := 'False'} : Bool := FALSE;   // Q896.2
      "Q896.3" { ExternalVisible := 'False'} : Bool := FALSE;   // Q896.3
      "Q896.4" { ExternalVisible := 'False'} : Bool := FALSE;   // Q896.4
      "Q896.5" { ExternalVisible := 'False'} : Bool := FALSE;   // Q896.5
      "Q896.6" { ExternalVisible := 'False'} : Bool := FALSE;   // Q896.6
      "Q896.7" { ExternalVisible := 'False'} : Bool := FALSE;   // Q896.7
      "Q897.0" { ExternalVisible := 'False'} : Bool := FALSE;   // Q897.0
      "Q897.1" { ExternalVisible := 'False'} : Bool := FALSE;   // Q897.1
      "Q897.2" { ExternalVisible := 'False'} : Bool := FALSE;   // Q897.2
      "Q897.3" { ExternalVisible := 'False'} : Bool := FALSE;   // Q897.3
      "Q897.4" { ExternalVisible := 'False'} : Bool := FALSE;   // Q897.4
      "Q897.5" { ExternalVisible := 'False'} : Bool := FALSE;   // Q897.5
      "Q897.6" { ExternalVisible := 'False'} : Bool := FALSE;   // Q897.6
      "Q897.7" { ExternalVisible := 'False'} : Bool := FALSE;   // Q897.7
      "Q898.0" { ExternalVisible := 'False'} : Bool := FALSE;   // Q898.0
      "Q898.1" { ExternalVisible := 'False'} : Bool := FALSE;   // Q898.1
      "Q898.2" { ExternalVisible := 'False'} : Bool := FALSE;   // Q898.2
      "Q898.3" { ExternalVisible := 'False'} : Bool := FALSE;   // Q898.3
      "Q898.4" { ExternalVisible := 'False'} : Bool := FALSE;   // Q898.4
      "Q898.5" { ExternalVisible := 'False'} : Bool := FALSE;   // Q898.5
      "Q898.6" { ExternalVisible := 'False'} : Bool := FALSE;   // Q898.6
      "Q898.7" { ExternalVisible := 'False'} : Bool := FALSE;   // Q898.7
      "Q899.0" { ExternalVisible := 'False'} : Bool := FALSE;   // Q899.0
      "Q899.1" { ExternalVisible := 'False'} : Bool := FALSE;   // Q899.1
      "Q899.2" { ExternalVisible := 'False'} : Bool := FALSE;   // Q899.2
      "Q899.3" { ExternalVisible := 'False'} : Bool := FALSE;   // Q899.3
      "Q899.4" { ExternalVisible := 'False'} : Bool := FALSE;   // Q899.4
      "Q899.5" { ExternalVisible := 'False'} : Bool := FALSE;   // Q899.5
      "Q899.6" { ExternalVisible := 'False'} : Bool := FALSE;   // Q899.6
      "Q899.7" { ExternalVisible := 'False'} : Bool := FALSE;   // Q899.7
      "Q900.0" { ExternalVisible := 'False'} : Bool := FALSE;   // Q900.0
      "Q900.1" { ExternalVisible := 'False'} : Bool := FALSE;   // Q900.1
      "Q900.2" { ExternalVisible := 'False'} : Bool := FALSE;   // Q900.2
      "Q900.3" { ExternalVisible := 'False'} : Bool := FALSE;   // Q900.3
      "Q900.4" { ExternalVisible := 'False'} : Bool := FALSE;   // Q900.4
      "Q900.5" { ExternalVisible := 'False'} : Bool := FALSE;   // Q900.5
      "Q900.6" { ExternalVisible := 'False'} : Bool := FALSE;   // Q900.6
      "Q900.7" { ExternalVisible := 'False'} : Bool := FALSE;   // Q900.7
   END_VAR
BEGIN
END_DATA_BLOCK

DATA_BLOCK "dGlobal"   // DB30150
{ S7_Optimized_Access := 'TRUE' }
// stored: AutoNumber false, MemoryReserve 100
   VAR
      gbo_Axis_Select { S7_SetPoint := 'True'} : Int;
      gbo_Pos_Select : Int;
      gto_Axis_Name : Array[0..9] of DB_ANY;
      gto_Axis_Index : DB_ANY;
      gr64_Pos_Index : LReal;
      Old_Axis_Select : Int;
      Old_Pos_Select : Int;
      gbo_Fault_Reset : Bool;
   END_VAR
   VAR RETAIN
      gi_Axis_AbsNum : Array[0..9] of Int;
   END_VAR
   VAR
      gbo_Axis_ManEnable : Array[0..9] of Bool;
   END_VAR
BEGIN
   gi_Axis_AbsNum[0] := 5;
   gi_Axis_AbsNum[1] := 6;
   gi_Axis_AbsNum[2] := 10;
   gi_Axis_AbsNum[3] := 5;
   gi_Axis_AbsNum[4] := 6;
   gi_Axis_AbsNum[5] := 7;
   gi_Axis_AbsNum[6] := 8;
   gi_Axis_AbsNum[7] := 9;
   gi_Axis_AbsNum[8..9] := 5;
   gbo_Axis_ManEnable[0..9] := 1;
END_DATA_BLOCK

DATA_BLOCK "dHMI"   // DB30151
{ S7_Optimized_Access := 'TRUE' }
// stored: AutoNumber false, MemoryReserve 100
   VAR
      HMI_SCREEN_Change : Array[1..4] of Int;
      HMI_SCREEN_NUM : Array[1..5] of Int;
   END_VAR
BEGIN
END_DATA_BLOCK

DATA_BLOCK "OneMES_ControlData"   // DB20230
{ S7_Optimized_Access := 'TRUE' }
// stored: AutoNumber false, MemoryReserve 100
   VAR
      HMI { S7_SetPoint := 'True'} : "UDT_OneMES_HMI_Control";
      MsgDisplay { S7_SetPoint := 'True'} : "UDT_MesMsgDisplay";
      Pluse { S7_SetPoint := 'True'} : Array[0..7] of Bool;
      OP : Array[1.."OP_Sum"] of "UDT_MESControl";
   END_VAR
BEGIN
   HMI.OP_Select := 1;
   HMI.PageCount := 1;
   // MsgDisplay.OP_Sel : 工站选择/暂不使用
   OP[1]."Timer"[1..15].PT := T#1s;
END_DATA_BLOCK

DATA_BLOCK "COLLECTIVE_SIGNAL_DB"   // DB117
{ S7_Optimized_Access := 'TRUE' }
// stored: MemoryReserve 100
   VAR
      COLLECTIVE_PD_ALARM : Bool;   // Collective signal: Alarms / Sammelsignal: Alarme
      COLLECTIVE_PD_WARNING : Bool;   // Collective signal: Warning / Sammelsignal: Warnungen
      COLLECTIVE_PD_INFO : Bool;   // Collective signal: Information / Sammelsignal: Information / Sammelsignal: 信息
      COLLECTIVE_SIGNAL_PD : USInt;   // 1: Alarm, 2: Warnung, 3: Information / 1: Alarm, 2: Warning, 3: Information / 1: 警报, 2: 警告, 3: 信息
   END_VAR
BEGIN
END_DATA_BLOCK

DATA_BLOCK "dStruct_Pos16"   // DB30141
{ S7_Optimized_Access := 'TRUE' }
// stored: AutoNumber false, MemoryReserve 100
   VAR
      Axis_Control_Data : Array[0..20] of Struct
         I_SS_bHome : Bool;   // 原点传感器
         I_SS_bFW : Bool;   // 前限位
         I_SS_bBW : Bool;   // 后限位
         I_CMD_bEnableAxis : Bool;   // 使能
         I_CMD_bResetAxis : Bool;   // 复位
         I_CMD_bjogForward : Bool;   // Taster Aufwärts / 正点
         I_CMD_bjogBackward : Bool;   // Taster Abwärts / 反点
         I_CMD_bmoveVelocity : Bool;   // 速度运行
         I_CMD_bstop : Bool;   // 停止
         I_CMD_bfastStop : Bool;   // 急停
         I_CMD_bHoming : Bool;   // 回零
         I_CMD_bGoToPos : Array[0..15] of Bool;   // Start Aufwärts in Automatik / 16个定位
         I_CMD_iGoToPos : Word;   // 16个定位 Word
         I_CMD_bCallAbsPos : Bool;   // 定位位置切换时，单独的定位按钮
         I_CMD_bRelPos : Bool;   // 相对定位
         I_CMD_MyBool : Array[0..5] of Bool;   // 临时变量
         I_Para_rJog_Speed : Array[0..2] of LReal;   // 点动速度/ACC/DEC/JERK
         I_Para_rMV_Speed : Array[0..2] of LReal;   // 速度运行速度/ACC/DEC/JERK
         I_Para_rStop_Dec : Array[0..1] of LReal;   // 速度运行速度/ACC/DEC/JERK
         I_Para_rEStop_Dec : Array[0..1] of LReal;   // 速度运行速度/ACC/DEC/JERK
         I_Para_iNum_Abspos : Int;
         I_Para_rPos_Abs : Array[0..16] of LReal;   // 绝对定位目标位置
         I_Para_rSpeed_Abs : Array[0..16] of LReal;   // Endlage Unten / 绝对定位速度
         I_Para_rAcc_Set : Array[0..16] of LReal;   // 绝对定位加速度
         I_Para_rDec_Set : Array[0..16] of LReal;   // 绝对定位减速度
         I_Para_rJerk_Set : Array[0..16] of LReal;   // 绝对定位加加速度
         I_Para_rSpeedPercent : LReal;   // Endlage Unten / 速度设定百分比
         I_Para_iHomeMode : Int;   // 回零方式
         I_Para_rHomePos : LReal;   // 回零位置
         O_Status_bAxisReady : Bool;   // 轴通讯正常
         O_Status_bAxisEnabled : Bool;   // 轴使能
         O_Status_bjogForward : Bool;   // 轴正点中
         O_Status_bjogBackward : Bool;   // 轴反点中
         O_Status_bHomed : Bool;   // 轴归零完成
         O_Status_bAtHome : Bool;   // 轴在零位
         O_Status_bSstill : Bool;   // 轴静止
         O_Status_bAxisBusy : Bool;   // 轴运行中
         O_Status_bAxisSyned : Bool;   // 同步上
         O_Status_bAxisError : Bool;   // 轴报警
         O_Status_bAtPos : Array[0..15] of Bool;   // Ausgang Aufwärts / 在目标位置上
         O_Status_bPosDone : Array[0..15] of Bool;   // 定位完成
         O_Status_bPosing : Array[0..15] of Bool;   // Ausgang Aufwärts / 定位中
         O_Status_bRelPosDone : Bool;   // 相对定位完成
         O_Status_rActPos : LReal;   // 实际位置
         O_Status_rActSpeed : LReal;   // 实际速度
         O_Status_iAxisFaultNum : UDInt;   // 轴报警代码
         O_Status_iDriveFaultNum : UDInt;   // 驱动报警代码
         O_Status_iFBStatus : Word;   // 运动功能块状态
         O_Status_iMCStatus : Word;   // 运动指令状态
         O_Status_rDriveTorque : LReal;   // 驱动扭矩
         O_Status_rDriveTemp : LReal;   // 驱动温度
         O_Status_rDriveRpm : LReal;   // 驱动转速
         O_Status_AxisName : WString[24];   // Name of axis
         O_Status_mybool : Array[0..5] of Bool;   // 备用
         O_Status_myLreal : Array[0..5] of LReal;   // 备用
         I_InLock_bEnableAxis : Bool;   // 使能
         I_InLock_bResetAxis : Bool;   // 复位
         I_InLock_bjogForward : Bool;   // Taster Aufwärts / 正点
         I_InLock_bjogBackward : Bool;   // Taster Abwärts / 反点
         I_InLock_bmoveVelocity : Bool;   // 速度运行
         I_InLock_bstop : Bool;   // 停止
         I_InLock_bfastStop : Bool;   // 急停
         I_InLock_bHoming : Bool;   // 回零
         I_InLock_bGoToPos : Array[0..16] of Bool;   // Start Aufwärts in Automatik / 16个定位
         I_InLock_iGoToPos : Word;   // 16个定位 Word
         I_InLock_bCallAbsPos : Bool;   // 定位位置切换时，单独的定位按钮
         I_InLock_bRelPos : Bool;   // 相对定位
         I_InLock_MyBool : Array[0..5] of Bool;   // 临时变量
         I_HMI_bEnableAxis : Bool;   // 使能
         I_HMI_bResetAxis : Bool;   // 复位
         I_HMI_bjogForward : Bool;   // Taster Aufwärts / 正点
         I_HMI_bjogBackward : Bool;   // Taster Abwärts / 反点
         I_HMI_bmoveVelocity : Bool;   // 速度运行
         I_HMI_bstop : Bool;   // 停止
         I_HMI_bfastStop : Bool;   // 急停
         I_HMI_bHoming : Bool;   // 回零
         I_HMI_bGoToPos : Array[0..16] of Bool;   // Start Aufwärts in Automatik / 16个定位
         I_HMI_iGoToPos : Word;   // 16个定位 Word
         I_HMI_bCallAbsPos : Bool;   // 定位位置切换时，单独的定位按钮
         I_HMI_bRelPos : Bool;   // 相对定位
         I_HMI_MyBool : Array[0..5] of Bool;   // 临时变量
         I_CDM_bGoToPos_0 : Bool;   // Start Aufwärts in Automatik / 16个定位自动
         I_InLock_bGoToPos_0 : Bool;   // Start Aufwärts in Automatik / 16个定位条件
         I_HMI_bGoToPos_0 : Bool;   // Start Aufwärts in Automatik / 16个定位HMI
         I_CDM_bGoToPos_1 : Bool;   // Start Aufwärts in Automatik / 16个定位自动
         I_InLock_bGoToPos_1 : Bool;   // Start Aufwärts in Automatik / 16个定位条件
         I_HMI_bGoToPos_1 : Bool;   // Start Aufwärts in Automatik / 16个定位HMI
         I_CDM_bGoToPos_2 : Bool;   // Start Aufwärts in Automatik / 16个定位自动
         I_InLock_bGoToPos_2 : Bool;   // Start Aufwärts in Automatik / 16个定位条件
         I_HMI_bGoToPos_2 : Bool;   // Start Aufwärts in Automatik / 16个定位HMI
         I_CDM_bGoToPos_3 : Bool;   // Start Aufwärts in Automatik / 16个定位自动
         I_InLock_bGoToPos_3 : Bool;   // Start Aufwärts in Automatik / 16个定位条件
         I_HMI_bGoToPos_3 : Bool;   // Start Aufwärts in Automatik / 16个定位HMI
         I_CDM_bGoToPos_4 : Bool;   // Start Aufwärts in Automatik / 16个定位自动
         I_InLock_bGoToPos_4 : Bool;   // Start Aufwärts in Automatik / 16个定位条件
         I_HMI_bGoToPos_4 : Bool;   // Start Aufwärts in Automatik / 16个定位HMI
         I_CDM_bGoToPos_5 : Bool;   // Start Aufwärts in Automatik / 16个定位自动
         I_InLock_bGoToPos_5 : Bool;   // Start Aufwärts in Automatik / 16个定位条件
         I_HMI_bGoToPos_5 : Bool;   // Start Aufwärts in Automatik / 16个定位HMI
         I_CDM_bGoToPos_6 : Bool;   // Start Aufwärts in Automatik / 16个定位自动
         I_InLock_bGoToPos_6 : Bool;   // Start Aufwärts in Automatik / 16个定位条件
         I_HMI_bGoToPos_6 : Bool;   // Start Aufwärts in Automatik / 16个定位HMI
         I_CDM_bGoToPos_7 : Bool;   // Start Aufwärts in Automatik / 16个定位自动
         I_InLock_bGoToPos_7 : Bool;   // Start Aufwärts in Automatik / 16个定位条件
         I_HMI_bGoToPos_7 : Bool;   // Start Aufwärts in Automatik / 16个定位HMI
         I_CDM_bGoToPos_8 : Bool;   // Start Aufwärts in Automatik / 16个定位自动
         I_InLock_bGoToPos_8 : Bool;   // Start Aufwärts in Automatik / 16个定位条件
         I_HMI_bGoToPos_8 : Bool;   // Start Aufwärts in Automatik / 16个定位HMI
      END_STRUCT;
      gs_AxisPos16 { S7_SetPoint := 'True'} : Array[0..9] of "sPos16";
   END_VAR
BEGIN
   Axis_Control_Data[0].I_SS_bFW := TRUE;
   Axis_Control_Data[0].I_SS_bBW := TRUE;
   Axis_Control_Data[0].I_Para_rJog_Speed[0] := 10.0;
   Axis_Control_Data[0].I_Para_rJog_Speed[1..2] := 30.0;
   Axis_Control_Data[0].I_Para_rMV_Speed[0] := 20.0;
   Axis_Control_Data[0].I_Para_rMV_Speed[1..2] := 30.0;
   Axis_Control_Data[0].I_Para_rStop_Dec[0] := 30.0;
   Axis_Control_Data[0].I_Para_rStop_Dec[1] := 50.0;
   Axis_Control_Data[0].I_Para_rEStop_Dec[0..1] := 50.0;
   Axis_Control_Data[0].I_Para_iNum_Abspos := 4;
   Axis_Control_Data[0].I_Para_rPos_Abs[1] := 10.0;
   Axis_Control_Data[0].I_Para_rPos_Abs[2] := 20.0;
   Axis_Control_Data[0].I_Para_rPos_Abs[3] := 30.0;
   Axis_Control_Data[0].I_Para_rPos_Abs[4] := 40.0;
   Axis_Control_Data[0].I_Para_rPos_Abs[5] := 50.0;
   Axis_Control_Data[0].I_Para_rPos_Abs[6] := 60.0;
   Axis_Control_Data[0].I_Para_rPos_Abs[7] := 70.0;
   Axis_Control_Data[0].I_Para_rPos_Abs[8] := 80.0;
   Axis_Control_Data[0].I_Para_rPos_Abs[9] := 90.0;
   Axis_Control_Data[0].I_Para_rPos_Abs[10] := 100.0;
   Axis_Control_Data[0].I_Para_rPos_Abs[11] := 110.0;
   Axis_Control_Data[0].I_Para_rPos_Abs[12] := 120.0;
   Axis_Control_Data[0].I_Para_rPos_Abs[13] := 130.0;
   Axis_Control_Data[0].I_Para_rPos_Abs[14] := 140.0;
   Axis_Control_Data[0].I_Para_rPos_Abs[15] := 150.0;
   Axis_Control_Data[0].I_Para_rPos_Abs[16] := 160.0;
   Axis_Control_Data[0].I_Para_rSpeed_Abs[0..16] := 20.0;
   Axis_Control_Data[0].I_Para_rAcc_Set[0..16] := 50.0;
   Axis_Control_Data[0].I_Para_rDec_Set[0..16] := 50.0;
   Axis_Control_Data[0].I_Para_rJerk_Set[0..16] := 50.0;
   Axis_Control_Data[0].I_Para_rSpeedPercent := 20.0;
   Axis_Control_Data[0].O_Status_AxisName := WSTRING#'No axis';
END_DATA_BLOCK

DATA_BLOCK "dStruct_Axis"   // DB30140
{ S7_Optimized_Access := 'TRUE' }
// stored: AutoNumber false, MemoryReserve 100
   VAR
      gs_Axis { S7_SetPoint := 'True'} : Array[0..9] of "sAxis";
      gs_Axis_HMI_Init { S7_SetPoint := 'True'} : "sAxis_HMI";
   END_VAR
BEGIN
END_DATA_BLOCK

ORGANIZATION_BLOCK "Main"   // OB1, LAD, ProgramCycle
TITLE = "Main Program Sweep (Cycle)"
{ S7_Optimized_Access := 'TRUE' }
// stored: SetENOAutomatically false
   VAR_INPUT
      Initial_Call : Bool;   // Initial call of this OB
      Remanence : Bool;   // =True, if remanent data are available
   END_VAR
BEGIN

REGION Network 1
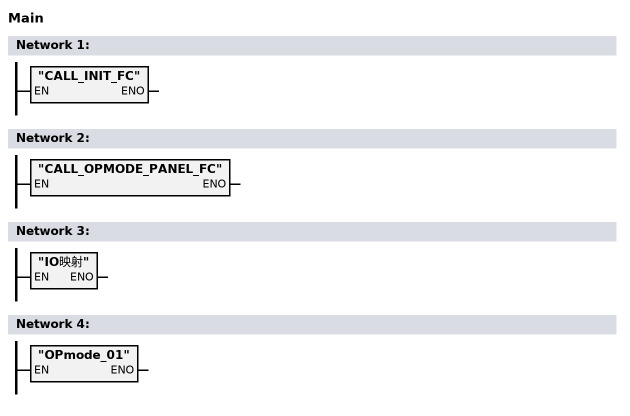
   RUNG wire#powerrail
      "CALL_INIT_FC"()
   END_RUNG
   // the same network as SCL:
   "CALL_INIT_FC"();
END_REGION

REGION Network 2
   RUNG wire#powerrail
      "CALL_OPMODE_PANEL_FC"()
   END_RUNG
   // the same network as SCL:
   "CALL_OPMODE_PANEL_FC"();
END_REGION

REGION Network 3
   RUNG wire#powerrail
      "IO映射"()
   END_RUNG
   // the same network as SCL:
   "IO映射"();
END_REGION

REGION Network 4
   RUNG wire#powerrail
      "OPmode_01"()
   END_RUNG
   // the same network as SCL:
   "OPmode_01"();
END_REGION
END_ORGANIZATION_BLOCK

FUNCTION "CALL_INIT_FC" : Void   // FC100, LAD
TITLE = Aufruf Initialisierung / Call initialization / Call 初始化
{ S7_Optimized_Access := 'TRUE' }
AUTHOR : Tesla
FAMILY : Base
VERSION : 1.0
// FUNKTIONSBESCHREIBUNG: 
// Der Baustein dient als Aufrufschnittstelle für die Bausteine, die einmalig bzgl. der Initialisierung aufgerufen werden müssen.
// Weitere Hinweise: siehe SICAR anwenderdefinierte Dokumentation / SICAR Online-Hilfe.
// DESCRIPTION OF FUNCTIONS:
// This function is the calling interface for initialization blocks.
// 描述 OF 功能:
// 这个 功能 is  calling 接口 给 初始化 blocks.
// stored: AutoNumber false, SetENOAutomatically false
BEGIN

REGION Network 1: Versorgung Globaler Informationen / Supply global information / 供应 全局 信息
   // 介绍：初始化功能，第一个被调用，调用一次，作用是定义OPMode和HMI数组长度，既最大数量，根据常数来决定。
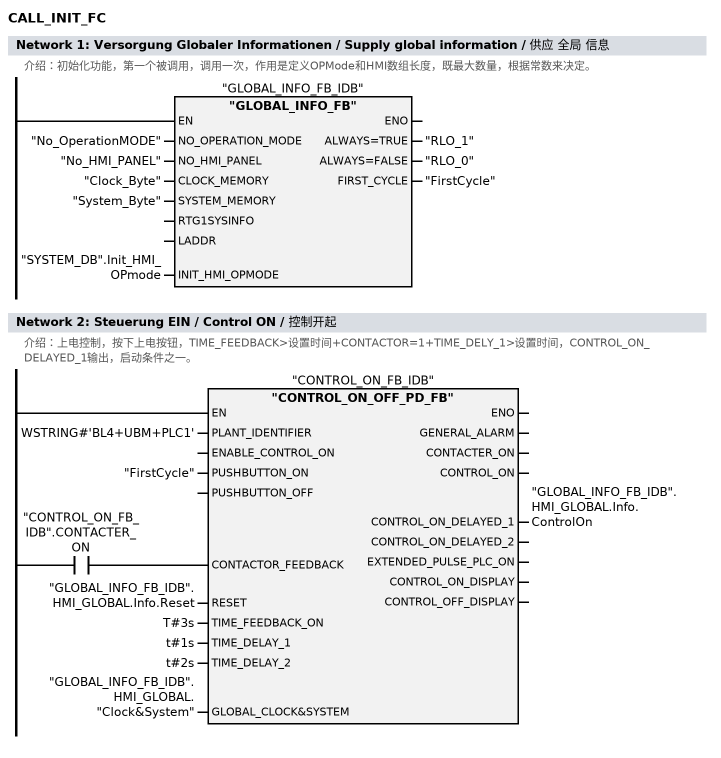
   RUNG wire#powerrail
      "GLOBAL_INFO_FB_IDB"(NO_OPERATION_MODE := "No_OperationMODE", NO_HMI_PANEL := "No_HMI_PANEL", CLOCK_MEMORY := "Clock_Byte", SYSTEM_MEMORY := "System_Byte", RTG1SYSINFO :=, LADDR :=, INIT_HMI_OPMODE := "SYSTEM_DB".Init_HMI_OPmode, "ALWAYS=TRUE" => "RLO_1", "ALWAYS=FALSE" => "RLO_0", FIRST_CYCLE => "FirstCycle")
   END_RUNG
   // the same network as SCL:
   "GLOBAL_INFO_FB_IDB"(NO_OPERATION_MODE := "No_OperationMODE",   // "GLOBAL_INFO_FB"
                        NO_HMI_PANEL := "No_HMI_PANEL",
                        CLOCK_MEMORY := "Clock_Byte",
                        SYSTEM_MEMORY := "System_Byte",
                        INIT_HMI_OPMODE := "SYSTEM_DB".Init_HMI_OPmode,
                        "ALWAYS=TRUE" => "RLO_1",
                        "ALWAYS=FALSE" => "RLO_0",
                        FIRST_CYCLE => "FirstCycle");
END_REGION

REGION Network 2: Steuerung EIN / Control ON / 控制开起
   // 介绍：上电控制，按下上电按钮，TIME_FEEDBACK>设置时间+CONTACTOR=1+TIME_DELY_1>设置时间，CONTROL_ON_DELAYED_1输出，启动条件之一。
   RUNG wire#powerrail
      "CONTROL_ON_FB_IDB"(CONTACTOR_FEEDBACK := wire#w1, PLANT_IDENTIFIER := WSTRING#'BL4+UBM+PLC1', ENABLE_CONTROL_ON :=, PUSHBUTTON_ON := "FirstCycle", PUSHBUTTON_OFF :=, RESET := "GLOBAL_INFO_FB_IDB".HMI_GLOBAL.Info.Reset, TIME_FEEDBACK_ON := T#3s, TIME_DELAY_1 := t#1s, TIME_DELAY_2 := t#2s, "GLOBAL_CLOCK&SYSTEM" := "GLOBAL_INFO_FB_IDB".HMI_GLOBAL."Clock&System", GENERAL_ALARM =>, CONTACTER_ON =>, CONTROL_ON =>, CONTROL_ON_DELAYED_1 => "GLOBAL_INFO_FB_IDB".HMI_GLOBAL.Info.ControlOn, CONTROL_ON_DELAYED_2 =>, EXTENDED_PULSE_PLC_ON =>, CONTROL_ON_DISPLAY =>, CONTROL_OFF_DISPLAY =>)
   END_RUNG
   RUNG wire#powerrail
      Contact( "CONTROL_ON_FB_IDB".CONTACTER_ON )
   END_RUNG wire#w1
   // the same network as SCL:
   "CONTROL_ON_FB_IDB"(PLANT_IDENTIFIER := WSTRING#'BL4+UBM+PLC1',   // "CONTROL_ON_OFF_PD_FB"
                       PUSHBUTTON_ON := "FirstCycle",
                       CONTACTOR_FEEDBACK := "CONTROL_ON_FB_IDB".CONTACTER_ON,
                       RESET := "GLOBAL_INFO_FB_IDB".HMI_GLOBAL.Info.Reset,
                       TIME_FEEDBACK_ON := T#3s,
                       TIME_DELAY_1 := t#1s,
                       TIME_DELAY_2 := t#2s,
                       "GLOBAL_CLOCK&SYSTEM" := "GLOBAL_INFO_FB_IDB".HMI_GLOBAL."Clock&System",
                       CONTROL_ON_DELAYED_1 => "GLOBAL_INFO_FB_IDB".HMI_GLOBAL.Info.ControlOn);
END_REGION
END_FUNCTION

FUNCTION "CALL_OPMODE_PANEL_FC" : Void   // FC200, LAD
TITLE = Aufruf Pult / Betriebsart / Call panels / operating modes
{ S7_Optimized_Access := 'TRUE' }
FAMILY : Base
VERSION : 1.0
// FUNKTIONSBESCHREIBUNG:
// Der Baustein dient als Aufrufschnittstelle für die HMI-/Panel- und Betriebsartenbausteine.
// Weitere Hinweise: siehe SICAR anwenderdefinierte Dokumentation / SICAR Online-Hilfe.
// DESCRIPTION OF FUNCTIONS:
// This function is the calling interface for initialization HMI/Panel and Operation mode blocks.
// For more informations see Tesla userdefined documentation / online-help.
// 描述 OF 功能:
// 这个 功能 is  calling 接口 给 初始化 HMI/Panel 和 运行 模式 blocks.
// 给 more informations see SICAR userdefined documentation / SICAR online-帮助.
// stored: AutoNumber false, SetENOAutomatically false
   VAR_TEMP
      Auxiliary_flag : Bool;
      Dummy_byte : Byte;
      dummy_word : Word;
      ParaAlarm : USInt;
      "020RB01_SlowDown" : Bool;
      "020RB02_SlowDown" : Bool;
      "020RB03_SlowDown" : Bool;
      "020RB04_SlowDown" : Bool;
      "020RB06_SlowDown" : Bool;
      "025RB01_SlowDown" : Bool;
      "025RB02_SlowDown" : Bool;
      "030RB01_SlowDown" : Bool;
      "030RB02_SlowDown" : Bool;
      "030RB03_SlowDown" : Bool;
      "030RB04_SlowDown" : Bool;
      待关联外部按钮1 : Bool;
      待关联外部按钮2 : Bool;
      待关联外部按钮2_1 : Bool;
   END_VAR
   VAR_TEMP   // added for the SCL form of the ladder/FBD networks
      _w1 : Bool;
      _w2 : Bool;
   END_VAR
BEGIN

REGION Network 1: Aufruf: HMI 1 / Call Operatorpanel_01: UBM1+010-HMI02 / Call: HMI_1
   // 介绍：设置和管理操作面板，
   // HMI:控制操作模式，可视化屏幕，
   // Panel：控制操作模式，按钮盒，
   // 有几个HMI调用几次，每次调用都需要对其定义类型。
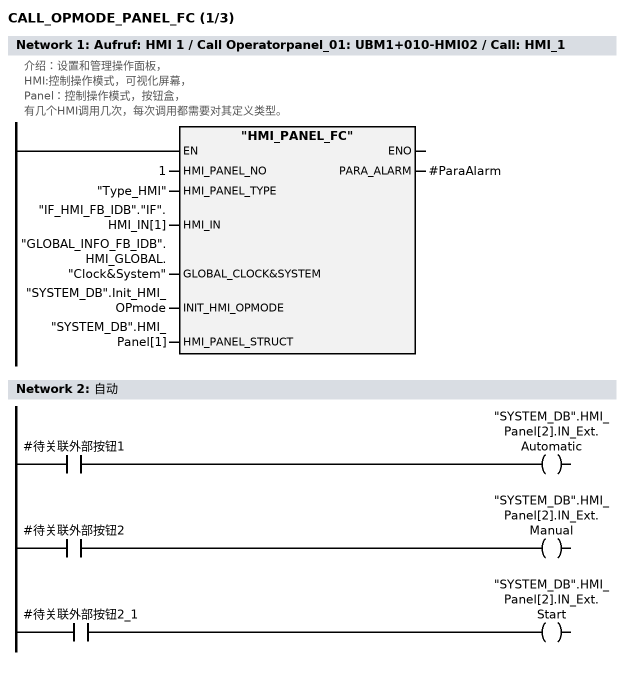
   RUNG wire#powerrail
      "HMI_PANEL_FC"(HMI_PANEL_NO := 1, HMI_PANEL_TYPE := "Type_HMI", HMI_IN := "IF_HMI_FB_IDB"."IF".HMI_IN[1], "GLOBAL_CLOCK&SYSTEM" := "GLOBAL_INFO_FB_IDB".HMI_GLOBAL."Clock&System", INIT_HMI_OPMODE := "SYSTEM_DB".Init_HMI_OPmode, HMI_PANEL_STRUCT := "SYSTEM_DB".HMI_Panel[1], PARA_ALARM => #ParaAlarm)
   END_RUNG
   // the same network as SCL:
   "HMI_PANEL_FC"(HMI_PANEL_NO := 1,
                  HMI_PANEL_TYPE := "Type_HMI",
                  HMI_IN := "IF_HMI_FB_IDB"."IF".HMI_IN[1],
                  "GLOBAL_CLOCK&SYSTEM" := "GLOBAL_INFO_FB_IDB".HMI_GLOBAL."Clock&System",
                  INIT_HMI_OPMODE := "SYSTEM_DB".Init_HMI_OPmode,
                  HMI_PANEL_STRUCT := "SYSTEM_DB".HMI_Panel[1],
                  PARA_ALARM => #ParaAlarm);
END_REGION

REGION Network 2: 自动
   RUNG wire#powerrail
      Contact( #待关联外部按钮1 )
      Coil( "SYSTEM_DB".HMI_Panel[2].IN_Ext.Automatic )
   END_RUNG
   RUNG wire#powerrail
      Contact( #待关联外部按钮2 )
      Coil( "SYSTEM_DB".HMI_Panel[2].IN_Ext.Manual )
   END_RUNG
   RUNG wire#powerrail
      Contact( #待关联外部按钮2_1 )
      Coil( "SYSTEM_DB".HMI_Panel[2].IN_Ext.Start )
   END_RUNG
   // the same network as SCL:
   "SYSTEM_DB".HMI_Panel[2].IN_Ext.Automatic := #待关联外部按钮1;
   "SYSTEM_DB".HMI_Panel[2].IN_Ext.Manual := #待关联外部按钮2;
   "SYSTEM_DB".HMI_Panel[2].IN_Ext.Start := #待关联外部按钮2_1;
END_REGION

